REGION Network 96: CONTADOR DE PRESENCIA - CNT_pHsMx_E1E3
   RUNG wire#powerrail
      #CNT_pHsMx_E1E3(IN := wire#w4, R := wire#w7, PV := #V_CNT_pHsMx_E1, BaseUnidades_ms := "CTE_BaseUnidades_1ms", QU =>, QD =>, CVU =>, CVD =>)
   END_RUNG
   RUNG wire#powerrail
      Contact( #Mx_ET10 )
      wire#w1
      Contact( #CNTSeg_pHsMx_E1E3.QU )
      wire#w2
      Contact( #Selec_M1_Entrada )
      Contact( #pHsMx_2 )
      wire#w3
      Contact( #Avance_E1_Tx_Ok )
      I_Contact( #EstadoZona.Manual_CBx )
   END_RUNG wire#w4
   RUNG wire#powerrail
      Contact( #Mx_ET51 )
      Contact( #Simultaneo_Mx )
   END_RUNG wire#w1
   RUNG wire#powerrail
      Contact( #Mx_ET11 )
   END_RUNG wire#w2
   RUNG wire#powerrail
      Contact( #Mx_ET12 )
   END_RUNG wire#w2
   RUNG wire#w2
      Contact( #Selec_M3_Entrada )
      Contact( #pHsMx_1 )
   END_RUNG wire#w3
   RUNG wire#powerrail
      I_Contact( #Mx_ET10 )
      wire#w5
      I_Contact( #Mx_ET11 )
      I_Contact( #Mx_ET12 )
      wire#w6
      I_Contact( #Mx_ET51 )
   END_RUNG wire#w7
   RUNG wire#powerrail
      I_Contact( #CNTSeg_pHsMx_E1E3.QU )
   END_RUNG wire#w5
   RUNG wire#w6
      I_Contact( #CNTSeg_pHsMx_E1E3.QU )
   END_RUNG wire#w7
   RUNG wire#w6
      I_Contact( #Simultaneo_Mx )
   END_RUNG wire#w7
   // the same network as SCL:
   #CNT_pHsMx_E1E3(IN := (((#Mx_ET10 OR (#Mx_ET51 AND #Simultaneo_Mx)) AND #CNTSeg_pHsMx_E1E3.QU) OR #Mx_ET11 OR #Mx_ET12) AND ((#Selec_M1_Entrada AND #pHsMx_2) OR (#Selec_M3_Entrada AND #pHsMx_1)) AND #Avance_E1_Tx_Ok AND NOT #EstadoZona.Manual_CBx,   // "FB910_CNT_UHS"
                   R := (NOT #Mx_ET10 OR NOT #CNTSeg_pHsMx_E1E3.QU) AND NOT #Mx_ET11 AND NOT #Mx_ET12 AND (NOT #Mx_ET51 OR NOT #CNTSeg_pHsMx_E1E3.QU OR NOT #Simultaneo_Mx),
                   PV := #V_CNT_pHsMx_E1,
                   BaseUnidades_ms := "CTE_BaseUnidades_1ms");
END_REGION

REGION Network 97: DETERMINA PASO ET10 - ET11 (Nota: Control de Tiempo para dar el FTF a la Mesa Anterior)
   RUNG wire#powerrail
      I_Contact( #Mx_ET00 )
      { S7_Templates := "SrcType := Int" } LE_Contact(in1 := #CNT_pHsMx_E1E3.CVD, in2 := #V_CNT_pHsMx_FTF_E1)
      { S7_Templates := "SrcType := Int" } LT_Contact(in1 := #CNT_pHsMx_E1E3.CVD, in2 := #V_CNT_pHsMx_E1)
      wire#w1
      Contact( #Selec_M1_Entrada )
      Contact( #pHsMx_2 )
      wire#w2
      Coil( #CNT_pHsMx_FTF_OK_E1E3 )
   END_RUNG
   RUNG wire#w1
      Contact( #Selec_M3_Entrada )
      Contact( #pHsMx_1 )
   END_RUNG wire#w2
   // the same network as SCL:
   #CNT_pHsMx_FTF_OK_E1E3 := NOT #Mx_ET00 AND (#CNT_pHsMx_E1E3.CVD <= #V_CNT_pHsMx_FTF_E1) AND (#CNT_pHsMx_E1E3.CVD < #V_CNT_pHsMx_E1) AND ((#Selec_M1_Entrada AND #pHsMx_2) OR (#Selec_M3_Entrada AND #pHsMx_1));
END_REGION

REGION Network 98: CONTADOR DE SEGURIDAD DE PRESENCIA - CNTSeg_pHsMx_E2E4
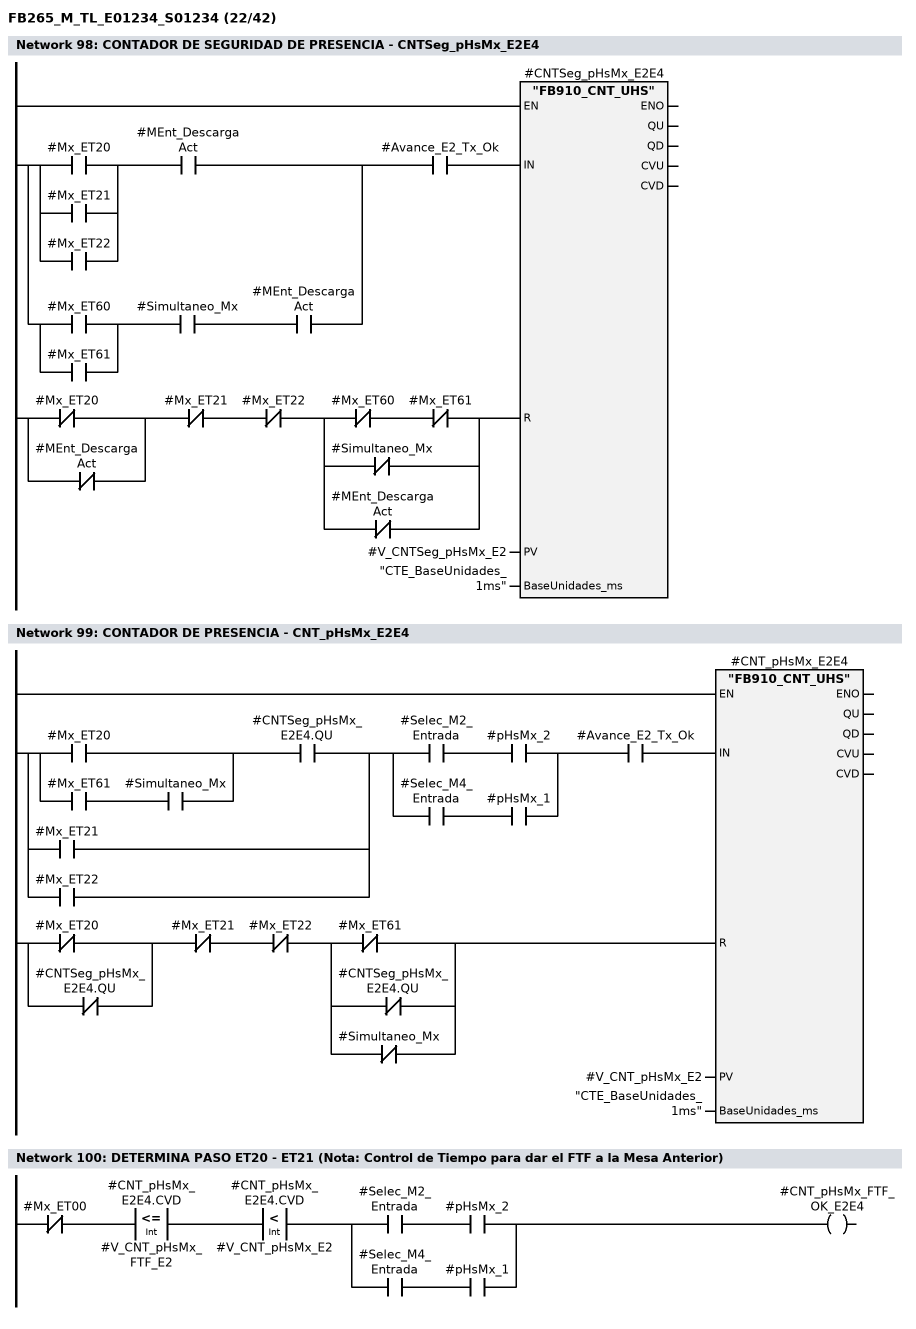
   RUNG wire#powerrail
      #CNTSeg_pHsMx_E2E4(IN := wire#w4, R := wire#w7, PV := #V_CNTSeg_pHsMx_E2, BaseUnidades_ms := "CTE_BaseUnidades_1ms", QU =>, QD =>, CVU =>, CVD =>)
   END_RUNG
   RUNG wire#powerrail
      Contact( #Mx_ET20 )
      wire#w1
      Contact( #MEnt_DescargaAct )
      wire#w2
      Contact( #Avance_E2_Tx_Ok )
   END_RUNG wire#w4
   RUNG wire#powerrail
      Contact( #Mx_ET21 )
   END_RUNG wire#w1
   RUNG wire#powerrail
      Contact( #Mx_ET22 )
   END_RUNG wire#w1
   RUNG wire#powerrail
      Contact( #Mx_ET60 )
      wire#w3
      Contact( #Simultaneo_Mx )
      Contact( #MEnt_DescargaAct )
   END_RUNG wire#w2
   RUNG wire#powerrail
      Contact( #Mx_ET61 )
   END_RUNG wire#w3
   RUNG wire#powerrail
      I_Contact( #Mx_ET20 )
      wire#w5
      I_Contact( #Mx_ET21 )
      I_Contact( #Mx_ET22 )
      wire#w6
      I_Contact( #Mx_ET60 )
      I_Contact( #Mx_ET61 )
   END_RUNG wire#w7
   RUNG wire#powerrail
      I_Contact( #MEnt_DescargaAct )
   END_RUNG wire#w5
   RUNG wire#w6
      I_Contact( #Simultaneo_Mx )
   END_RUNG wire#w7
   RUNG wire#w6
      I_Contact( #MEnt_DescargaAct )
   END_RUNG wire#w7
   // the same network as SCL:
   #CNTSeg_pHsMx_E2E4(IN := (((#Mx_ET20 OR #Mx_ET21 OR #Mx_ET22) AND #MEnt_DescargaAct) OR ((#Mx_ET60 OR #Mx_ET61) AND #Simultaneo_Mx AND #MEnt_DescargaAct)) AND #Avance_E2_Tx_Ok,   // "FB910_CNT_UHS"
                      R := (NOT #Mx_ET20 OR NOT #MEnt_DescargaAct) AND NOT #Mx_ET21 AND NOT #Mx_ET22 AND ((NOT #Mx_ET60 AND NOT #Mx_ET61) OR NOT #Simultaneo_Mx OR NOT #MEnt_DescargaAct),
                      PV := #V_CNTSeg_pHsMx_E2,
                      BaseUnidades_ms := "CTE_BaseUnidades_1ms");
END_REGION

REGION Network 99: CONTADOR DE PRESENCIA - CNT_pHsMx_E2E4
   RUNG wire#powerrail
      #CNT_pHsMx_E2E4(IN := wire#w4, R := wire#w7, PV := #V_CNT_pHsMx_E2, BaseUnidades_ms := "CTE_BaseUnidades_1ms", QU =>, QD =>, CVU =>, CVD =>)
   END_RUNG
   RUNG wire#powerrail
      Contact( #Mx_ET20 )
      wire#w1
      Contact( #CNTSeg_pHsMx_E2E4.QU )
      wire#w2
      Contact( #Selec_M2_Entrada )
      Contact( #pHsMx_2 )
      wire#w3
      Contact( #Avance_E2_Tx_Ok )
   END_RUNG wire#w4
   RUNG wire#powerrail
      Contact( #Mx_ET61 )
      Contact( #Simultaneo_Mx )
   END_RUNG wire#w1
   RUNG wire#powerrail
      Contact( #Mx_ET21 )
   END_RUNG wire#w2
   RUNG wire#powerrail
      Contact( #Mx_ET22 )
   END_RUNG wire#w2
   RUNG wire#w2
      Contact( #Selec_M4_Entrada )
      Contact( #pHsMx_1 )
   END_RUNG wire#w3
   RUNG wire#powerrail
      I_Contact( #Mx_ET20 )
      wire#w5
      I_Contact( #Mx_ET21 )
      I_Contact( #Mx_ET22 )
      wire#w6
      I_Contact( #Mx_ET61 )
   END_RUNG wire#w7
   RUNG wire#powerrail
      I_Contact( #CNTSeg_pHsMx_E2E4.QU )
   END_RUNG wire#w5
   RUNG wire#w6
      I_Contact( #CNTSeg_pHsMx_E2E4.QU )
   END_RUNG wire#w7
   RUNG wire#w6
      I_Contact( #Simultaneo_Mx )
   END_RUNG wire#w7
   // the same network as SCL:
   #CNT_pHsMx_E2E4(IN := (((#Mx_ET20 OR (#Mx_ET61 AND #Simultaneo_Mx)) AND #CNTSeg_pHsMx_E2E4.QU) OR #Mx_ET21 OR #Mx_ET22) AND ((#Selec_M2_Entrada AND #pHsMx_2) OR (#Selec_M4_Entrada AND #pHsMx_1)) AND #Avance_E2_Tx_Ok,   // "FB910_CNT_UHS"
                   R := (NOT #Mx_ET20 OR NOT #CNTSeg_pHsMx_E2E4.QU) AND NOT #Mx_ET21 AND NOT #Mx_ET22 AND (NOT #Mx_ET61 OR NOT #CNTSeg_pHsMx_E2E4.QU OR NOT #Simultaneo_Mx),
                   PV := #V_CNT_pHsMx_E2,
                   BaseUnidades_ms := "CTE_BaseUnidades_1ms");
END_REGION

REGION Network 100: DETERMINA PASO ET20 - ET21 (Nota: Control de Tiempo para dar el FTF a la Mesa Anterior)
   RUNG wire#powerrail
      I_Contact( #Mx_ET00 )
      { S7_Templates := "SrcType := Int" } LE_Contact(in1 := #CNT_pHsMx_E2E4.CVD, in2 := #V_CNT_pHsMx_FTF_E2)
      { S7_Templates := "SrcType := Int" } LT_Contact(in1 := #CNT_pHsMx_E2E4.CVD, in2 := #V_CNT_pHsMx_E2)
      wire#w1
      Contact( #Selec_M2_Entrada )
      Contact( #pHsMx_2 )
      wire#w2
      Coil( #CNT_pHsMx_FTF_OK_E2E4 )
   END_RUNG
   RUNG wire#w1
      Contact( #Selec_M4_Entrada )
      Contact( #pHsMx_1 )
   END_RUNG wire#w2
   // the same network as SCL:
   #CNT_pHsMx_FTF_OK_E2E4 := NOT #Mx_ET00 AND (#CNT_pHsMx_E2E4.CVD <= #V_CNT_pHsMx_FTF_E2) AND (#CNT_pHsMx_E2E4.CVD < #V_CNT_pHsMx_E2) AND ((#Selec_M2_Entrada AND #pHsMx_2) OR (#Selec_M4_Entrada AND #pHsMx_1));
END_REGION

REGION Network 101: CONTADOR SEGURIDAD DE AUSENCIA - CNTSeg_ApHsMx ??????? RESTAR VALOR DE POSICIONAMIENTO
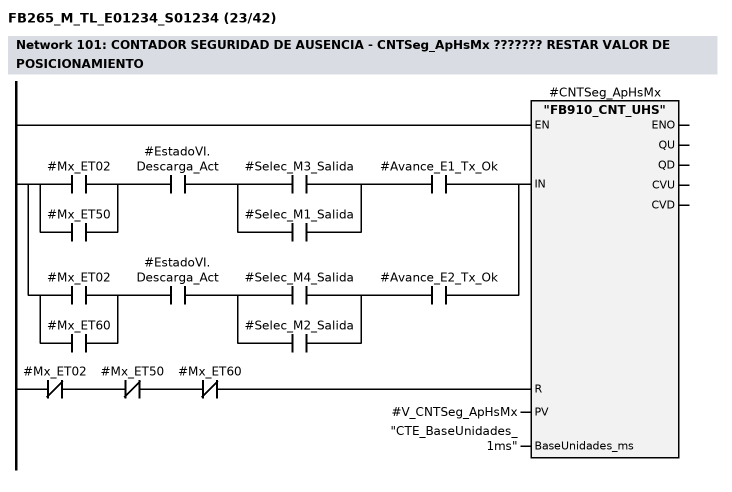
   RUNG wire#powerrail
      #CNTSeg_ApHsMx(IN := wire#w7, R := wire#w8, PV := #V_CNTSeg_ApHsMx, BaseUnidades_ms := "CTE_BaseUnidades_1ms", QU =>, QD =>, CVU =>, CVD =>)
   END_RUNG
   RUNG wire#powerrail
      Contact( #Mx_ET02 )
      wire#w1
      Contact( #EstadoVI.Descarga_Act )
      wire#w2
      Contact( #Selec_M3_Salida )
      wire#w3
      Contact( #Avance_E1_Tx_Ok )
   END_RUNG wire#w7
   RUNG wire#powerrail
      Contact( #Mx_ET50 )
   END_RUNG wire#w1
   RUNG wire#w2
      Contact( #Selec_M1_Salida )
   END_RUNG wire#w3
   RUNG wire#powerrail
      Contact( #Mx_ET02 )
      wire#w4
      Contact( #EstadoVI.Descarga_Act )
      wire#w5
      Contact( #Selec_M4_Salida )
      wire#w6
      Contact( #Avance_E2_Tx_Ok )
   END_RUNG wire#w7
   RUNG wire#powerrail
      Contact( #Mx_ET60 )
   END_RUNG wire#w4
   RUNG wire#w5
      Contact( #Selec_M2_Salida )
   END_RUNG wire#w6
   RUNG wire#powerrail
      I_Contact( #Mx_ET02 )
      I_Contact( #Mx_ET50 )
      I_Contact( #Mx_ET60 )
   END_RUNG wire#w8
   // the same network as SCL:
   #CNTSeg_ApHsMx(IN := ((#Mx_ET02 OR #Mx_ET50) AND #EstadoVI.Descarga_Act AND (#Selec_M3_Salida OR #Selec_M1_Salida) AND #Avance_E1_Tx_Ok) OR ((#Mx_ET02 OR #Mx_ET60) AND #EstadoVI.Descarga_Act AND (#Selec_M4_Salida OR #Selec_M2_Salida) AND #Avance_E2_Tx_Ok),   // "FB910_CNT_UHS"
                  R := NOT #Mx_ET02 AND NOT #Mx_ET50 AND NOT #Mx_ET60,
                  PV := #V_CNTSeg_ApHsMx,
                  BaseUnidades_ms := "CTE_BaseUnidades_1ms");
END_REGION

REGION Network 102: CONTADOR DE LA AUSENCIA - CNT_ApHsMX
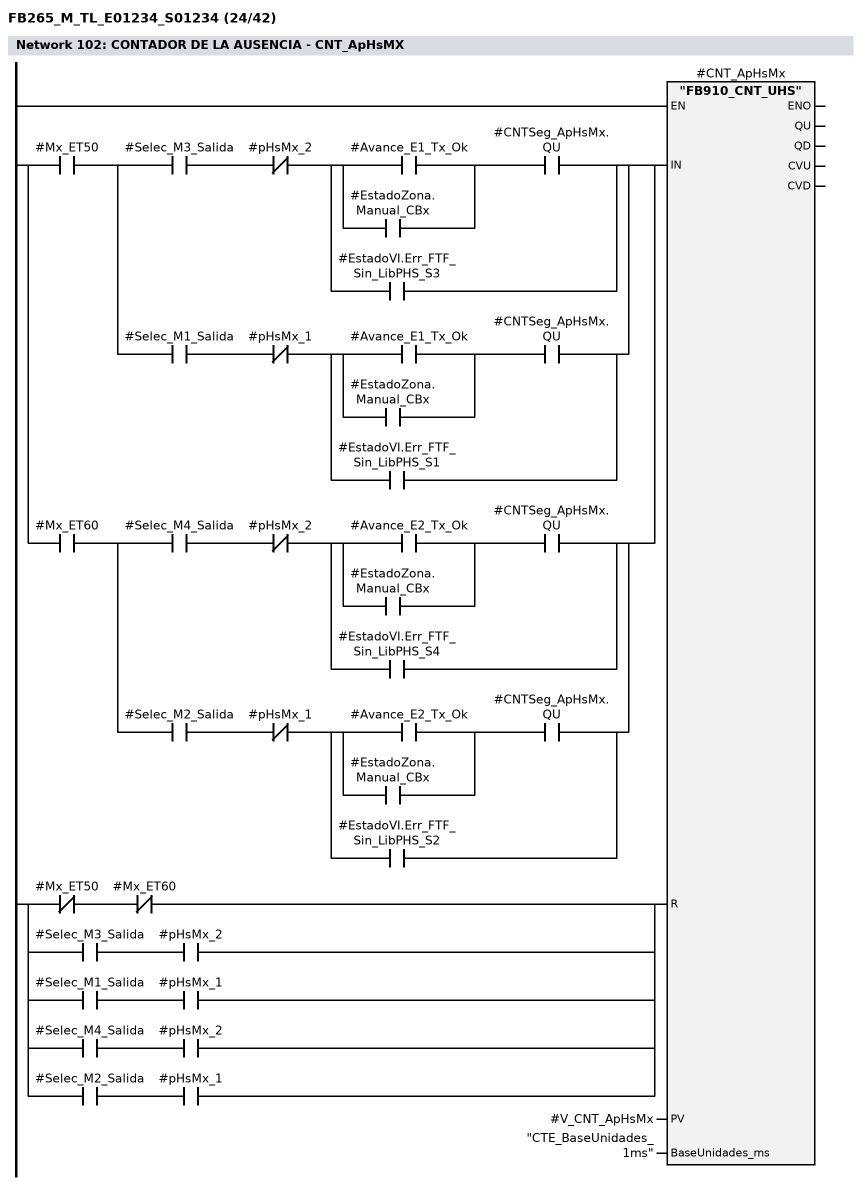
   RUNG wire#powerrail
      #CNT_ApHsMx(IN := wire#w11, R := wire#w12, PV := #V_CNT_ApHsMx, BaseUnidades_ms := "CTE_BaseUnidades_1ms", QU =>, QD =>, CVU =>, CVD =>)
   END_RUNG
   RUNG wire#powerrail
      Contact( #Mx_ET50 )
      wire#w1
      Contact( #Selec_M3_Salida )
      I_Contact( #pHsMx_2 )
      wire#w2
      Contact( #Avance_E1_Tx_Ok )
      wire#w3
      Contact( #CNTSeg_ApHsMx.QU )
   END_RUNG wire#w11
   RUNG wire#w2
      Contact( #EstadoZona.Manual_CBx )
   END_RUNG wire#w3
   RUNG wire#w2
      Contact( #EstadoVI.Err_FTF_Sin_LibPHS_S3 )
   END_RUNG wire#w11
   RUNG wire#w1
      Contact( #Selec_M1_Salida )
      I_Contact( #pHsMx_1 )
      wire#w4
      Contact( #Avance_E1_Tx_Ok )
      wire#w5
      Contact( #CNTSeg_ApHsMx.QU )
   END_RUNG wire#w11
   RUNG wire#w4
      Contact( #EstadoZona.Manual_CBx )
   END_RUNG wire#w5
   RUNG wire#w4
      Contact( #EstadoVI.Err_FTF_Sin_LibPHS_S1 )
   END_RUNG wire#w11
   RUNG wire#powerrail
      Contact( #Mx_ET60 )
      wire#w6
      Contact( #Selec_M4_Salida )
      I_Contact( #pHsMx_2 )
      wire#w7
      Contact( #Avance_E2_Tx_Ok )
      wire#w8
      Contact( #CNTSeg_ApHsMx.QU )
   END_RUNG wire#w11
   RUNG wire#w7
      Contact( #EstadoZona.Manual_CBx )
   END_RUNG wire#w8
   RUNG wire#w7
      Contact( #EstadoVI.Err_FTF_Sin_LibPHS_S4 )
   END_RUNG wire#w11
   RUNG wire#w6
      Contact( #Selec_M2_Salida )
      I_Contact( #pHsMx_1 )
      wire#w9
      Contact( #Avance_E2_Tx_Ok )
      wire#w10
      Contact( #CNTSeg_ApHsMx.QU )
   END_RUNG wire#w11
   RUNG wire#w9
      Contact( #EstadoZona.Manual_CBx )
   END_RUNG wire#w10
   RUNG wire#w9
      Contact( #EstadoVI.Err_FTF_Sin_LibPHS_S2 )
   END_RUNG wire#w11
   RUNG wire#powerrail
      I_Contact( #Mx_ET50 )
      I_Contact( #Mx_ET60 )
   END_RUNG wire#w12
   RUNG wire#powerrail
      Contact( #Selec_M3_Salida )
      Contact( #pHsMx_2 )
   END_RUNG wire#w12
   RUNG wire#powerrail
      Contact( #Selec_M1_Salida )
      Contact( #pHsMx_1 )
   END_RUNG wire#w12
   RUNG wire#powerrail
      Contact( #Selec_M4_Salida )
      Contact( #pHsMx_2 )
   END_RUNG wire#w12
   RUNG wire#powerrail
      Contact( #Selec_M2_Salida )
      Contact( #pHsMx_1 )
   END_RUNG wire#w12
   // the same network as SCL:
   #CNT_ApHsMx(IN := (#Mx_ET50 AND ((#Selec_M3_Salida AND NOT #pHsMx_2 AND (((#Avance_E1_Tx_Ok OR #EstadoZona.Manual_CBx) AND #CNTSeg_ApHsMx.QU) OR #EstadoVI.Err_FTF_Sin_LibPHS_S3)) OR (#Selec_M1_Salida AND NOT #pHsMx_1 AND (((#Avance_E1_Tx_Ok OR #EstadoZona.Manual_CBx) AND #CNTSeg_ApHsMx.QU) OR #EstadoVI.Err_FTF_Sin_LibPHS_S1)))) OR (#Mx_ET60 AND ((#Selec_M4_Salida AND NOT #pHsMx_2 AND (((#Avance_E2_Tx_Ok OR #EstadoZona.Manual_CBx) AND #CNTSeg_ApHsMx.QU) OR #EstadoVI.Err_FTF_Sin_LibPHS_S4)) OR (#Selec_M2_Salida AND NOT #pHsMx_1 AND (((#Avance_E2_Tx_Ok OR #EstadoZona.Manual_CBx) AND #CNTSeg_ApHsMx.QU) OR #EstadoVI.Err_FTF_Sin_LibPHS_S2)))),   // "FB910_CNT_UHS"
               R := (NOT #Mx_ET50 AND NOT #Mx_ET60) OR (#Selec_M3_Salida AND #pHsMx_2) OR (#Selec_M1_Salida AND #pHsMx_1) OR (#Selec_M4_Salida AND #pHsMx_2) OR (#Selec_M2_Salida AND #pHsMx_1),
               PV := #V_CNT_ApHsMx,
               BaseUnidades_ms := "CTE_BaseUnidades_1ms");
END_REGION

REGION Network 103: TEMPORIZADOR DE BLOQUEO DE MESA
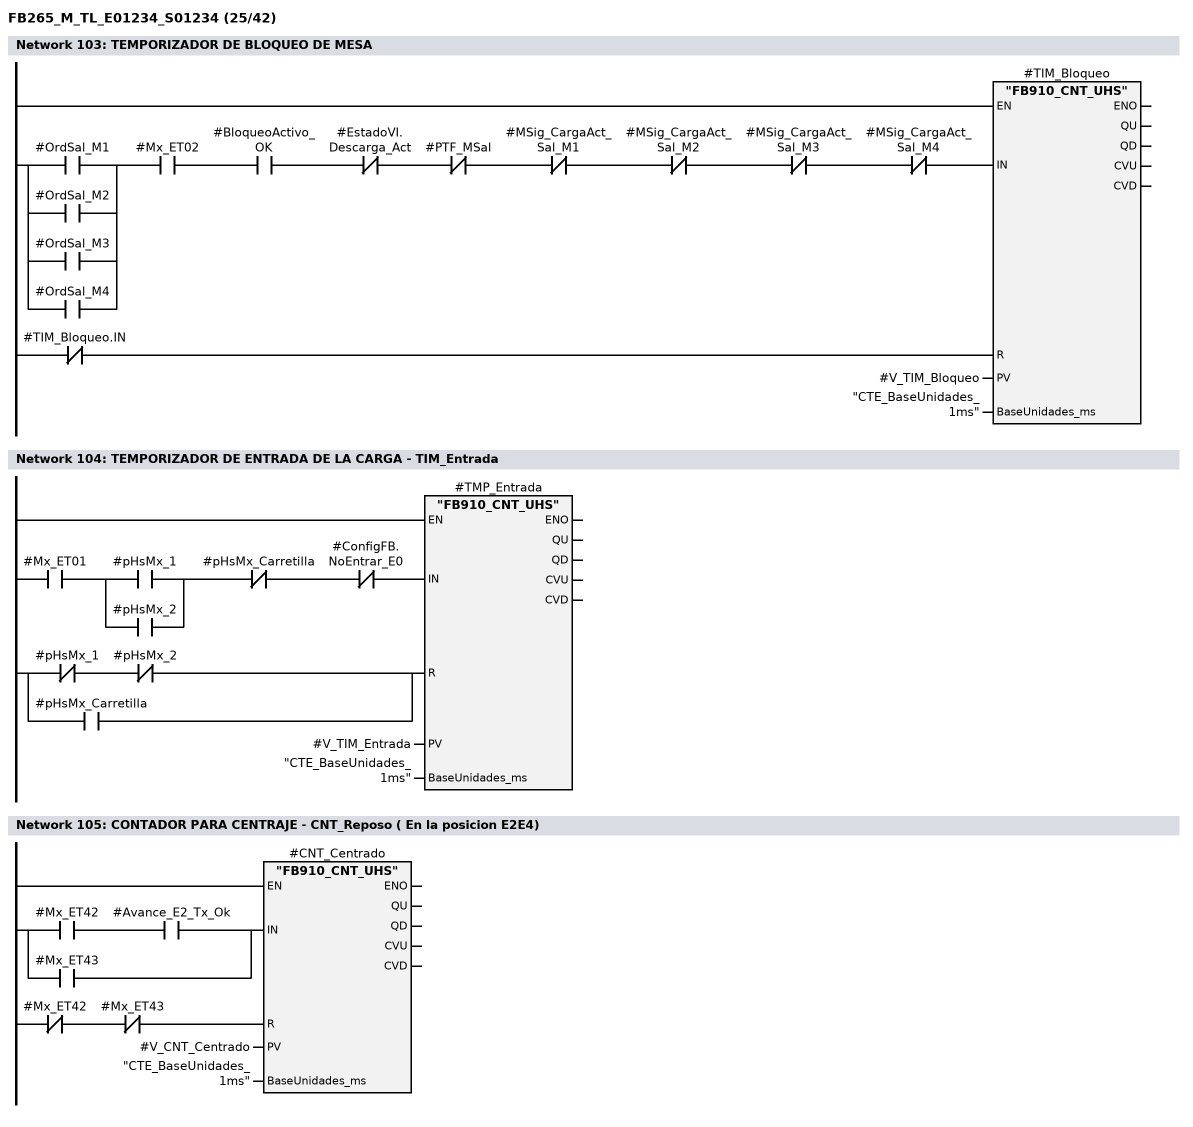
   RUNG wire#powerrail
      #TIM_Bloqueo(IN := wire#w2, R := wire#w3, PV := #V_TIM_Bloqueo, BaseUnidades_ms := "CTE_BaseUnidades_1ms", QU =>, QD =>, CVU =>, CVD =>)
   END_RUNG
   RUNG wire#powerrail
      Contact( #OrdSal_M1 )
      wire#w1
      Contact( #Mx_ET02 )
      Contact( #BloqueoActivo_OK )
      I_Contact( #EstadoVI.Descarga_Act )
      I_Contact( #PTF_MSal )
      I_Contact( #MSig_CargaAct_Sal_M1 )
      I_Contact( #MSig_CargaAct_Sal_M2 )
      I_Contact( #MSig_CargaAct_Sal_M3 )
      I_Contact( #MSig_CargaAct_Sal_M4 )
   END_RUNG wire#w2
   RUNG wire#powerrail
      Contact( #OrdSal_M2 )
   END_RUNG wire#w1
   RUNG wire#powerrail
      Contact( #OrdSal_M3 )
   END_RUNG wire#w1
   RUNG wire#powerrail
      Contact( #OrdSal_M4 )
   END_RUNG wire#w1
   RUNG wire#powerrail
      I_Contact( #TIM_Bloqueo.IN )
   END_RUNG wire#w3
   // the same network as SCL:
   #TIM_Bloqueo(IN := (#OrdSal_M1 OR #OrdSal_M2 OR #OrdSal_M3 OR #OrdSal_M4) AND #Mx_ET02 AND #BloqueoActivo_OK AND NOT #EstadoVI.Descarga_Act AND NOT #PTF_MSal AND NOT #MSig_CargaAct_Sal_M1 AND NOT #MSig_CargaAct_Sal_M2 AND NOT #MSig_CargaAct_Sal_M3 AND NOT #MSig_CargaAct_Sal_M4,   // "FB910_CNT_UHS"
                R := NOT #TIM_Bloqueo.IN,
                PV := #V_TIM_Bloqueo,
                BaseUnidades_ms := "CTE_BaseUnidades_1ms");
END_REGION

REGION Network 104: TEMPORIZADOR DE ENTRADA DE LA CARGA - TIM_Entrada
   RUNG wire#powerrail
      #TMP_Entrada(IN := wire#w3, R := wire#w4, PV := #V_TIM_Entrada, BaseUnidades_ms := "CTE_BaseUnidades_1ms", QU =>, QD =>, CVU =>, CVD =>)
   END_RUNG
   RUNG wire#powerrail
      Contact( #Mx_ET01 )
      wire#w1
      Contact( #pHsMx_1 )
      wire#w2
      I_Contact( #pHsMx_Carretilla )
      I_Contact( #ConfigFB.NoEntrar_E0 )
   END_RUNG wire#w3
   RUNG wire#w1
      Contact( #pHsMx_2 )
   END_RUNG wire#w2
   RUNG wire#powerrail
      I_Contact( #pHsMx_1 )
      I_Contact( #pHsMx_2 )
   END_RUNG wire#w4
   RUNG wire#powerrail
      Contact( #pHsMx_Carretilla )
   END_RUNG wire#w4
   // the same network as SCL:
   #TMP_Entrada(IN := #Mx_ET01 AND (#pHsMx_1 OR #pHsMx_2) AND NOT #pHsMx_Carretilla AND NOT #ConfigFB.NoEntrar_E0,   // "FB910_CNT_UHS"
                R := (NOT #pHsMx_1 AND NOT #pHsMx_2) OR #pHsMx_Carretilla,
                PV := #V_TIM_Entrada,
                BaseUnidades_ms := "CTE_BaseUnidades_1ms");
END_REGION

REGION Network 105: CONTADOR PARA CENTRAJE - CNT_Reposo ( En la posicion E2E4)
   RUNG wire#powerrail
      #CNT_Centrado(IN := wire#w1, R := wire#w2, PV := #V_CNT_Centrado, BaseUnidades_ms := "CTE_BaseUnidades_1ms", QU =>, QD =>, CVU =>, CVD =>)
   END_RUNG
   RUNG wire#powerrail
      Contact( #Mx_ET42 )
      Contact( #Avance_E2_Tx_Ok )
   END_RUNG wire#w1
   RUNG wire#powerrail
      Contact( #Mx_ET43 )
   END_RUNG wire#w1
   RUNG wire#powerrail
      I_Contact( #Mx_ET42 )
      I_Contact( #Mx_ET43 )
   END_RUNG wire#w2
   // the same network as SCL:
   #CNT_Centrado(IN := (#Mx_ET42 AND #Avance_E2_Tx_Ok) OR #Mx_ET43,   // "FB910_CNT_UHS"
                 R := NOT #Mx_ET42 AND NOT #Mx_ET43,
                 PV := #V_CNT_Centrado,
                 BaseUnidades_ms := "CTE_BaseUnidades_1ms");
END_REGION

REGION Network 106: TEMPORIZADOR DE RETIRADA DE LA CARGA - TIM_Salida
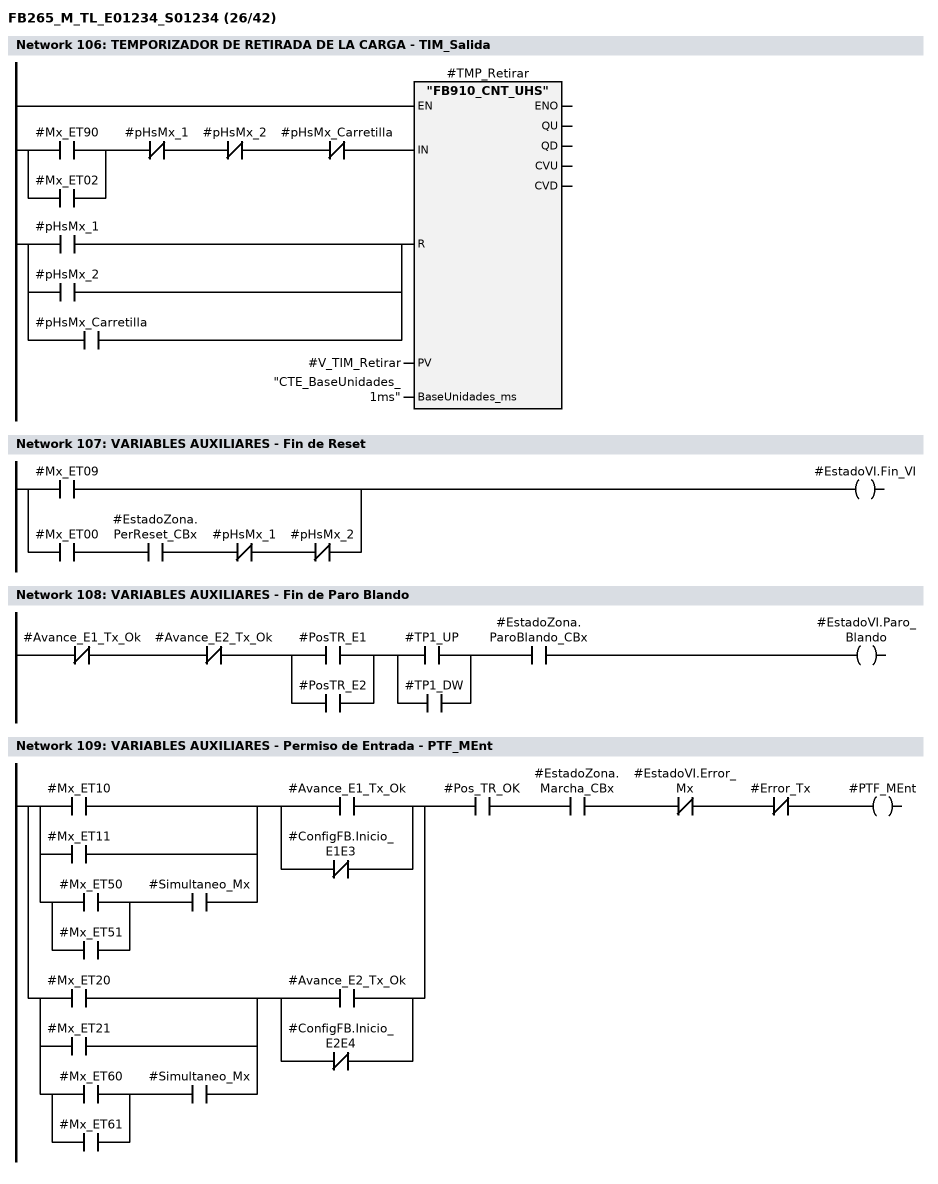
   RUNG wire#powerrail
      #TMP_Retirar(IN := wire#w2, R := wire#w3, PV := #V_TIM_Retirar, BaseUnidades_ms := "CTE_BaseUnidades_1ms", QU =>, QD =>, CVU =>, CVD =>)
   END_RUNG
   RUNG wire#powerrail
      Contact( #Mx_ET90 )
      wire#w1
      I_Contact( #pHsMx_1 )
      I_Contact( #pHsMx_2 )
      I_Contact( #pHsMx_Carretilla )
   END_RUNG wire#w2
   RUNG wire#powerrail
      Contact( #Mx_ET02 )
   END_RUNG wire#w1
   RUNG wire#powerrail
      Contact( #pHsMx_1 )
   END_RUNG wire#w3
   RUNG wire#powerrail
      Contact( #pHsMx_2 )
   END_RUNG wire#w3
   RUNG wire#powerrail
      Contact( #pHsMx_Carretilla )
   END_RUNG wire#w3
   // the same network as SCL:
   #TMP_Retirar(IN := (#Mx_ET90 OR #Mx_ET02) AND NOT #pHsMx_1 AND NOT #pHsMx_2 AND NOT #pHsMx_Carretilla,   // "FB910_CNT_UHS"
                R := #pHsMx_1 OR #pHsMx_2 OR #pHsMx_Carretilla,
                PV := #V_TIM_Retirar,
                BaseUnidades_ms := "CTE_BaseUnidades_1ms");
END_REGION

REGION Network 107: VARIABLES AUXILIARES - Fin de Reset
   RUNG wire#powerrail
      Contact( #Mx_ET09 )
      wire#w1
      Coil( #EstadoVI.Fin_VI )
   END_RUNG
   RUNG wire#powerrail
      Contact( #Mx_ET00 )
      Contact( #EstadoZona.PerReset_CBx )
      I_Contact( #pHsMx_1 )
      I_Contact( #pHsMx_2 )
   END_RUNG wire#w1
   // the same network as SCL:
   #EstadoVI.Fin_VI := #Mx_ET09 OR (#Mx_ET00 AND #EstadoZona.PerReset_CBx AND NOT #pHsMx_1 AND NOT #pHsMx_2);
END_REGION

REGION Network 108: VARIABLES AUXILIARES - Fin de Paro Blando
   RUNG wire#powerrail
      I_Contact( #Avance_E1_Tx_Ok )
      I_Contact( #Avance_E2_Tx_Ok )
      wire#w1
      Contact( #PosTR_E1 )
      wire#w2
      Contact( #TP1_UP )
      wire#w3
      Contact( #EstadoZona.ParoBlando_CBx )
      Coil( #EstadoVI.Paro_Blando )
   END_RUNG
   RUNG wire#w1
      Contact( #PosTR_E2 )
   END_RUNG wire#w2
   RUNG wire#w2
      Contact( #TP1_DW )
   END_RUNG wire#w3
   // the same network as SCL:
   #EstadoVI.Paro_Blando := NOT #Avance_E1_Tx_Ok AND NOT #Avance_E2_Tx_Ok AND (#PosTR_E1 OR #PosTR_E2) AND (#TP1_UP OR #TP1_DW) AND #EstadoZona.ParoBlando_CBx;
END_REGION

REGION Network 109: VARIABLES AUXILIARES - Permiso de Entrada - PTF_MEnt
   RUNG wire#powerrail
      Contact( #Mx_ET10 )
      wire#w1
      Contact( #Avance_E1_Tx_Ok )
      wire#w3
      Contact( #Pos_TR_OK )
      Contact( #EstadoZona.Marcha_CBx )
      I_Contact( #EstadoVI.Error_Mx )
      I_Contact( #Error_Tx )
      Coil( #PTF_MEnt )
   END_RUNG
   RUNG wire#powerrail
      Contact( #Mx_ET11 )
   END_RUNG wire#w1
   RUNG wire#powerrail
      Contact( #Mx_ET50 )
      wire#w2
      Contact( #Simultaneo_Mx )
   END_RUNG wire#w1
   RUNG wire#powerrail
      Contact( #Mx_ET51 )
   END_RUNG wire#w2
   RUNG wire#w1
      I_Contact( #ConfigFB.Inicio_E1E3 )
   END_RUNG wire#w3
   RUNG wire#powerrail
      Contact( #Mx_ET20 )
      wire#w4
      Contact( #Avance_E2_Tx_Ok )
   END_RUNG wire#w3
   RUNG wire#powerrail
      Contact( #Mx_ET21 )
   END_RUNG wire#w4
   RUNG wire#powerrail
      Contact( #Mx_ET60 )
      wire#w5
      Contact( #Simultaneo_Mx )
   END_RUNG wire#w4
   RUNG wire#powerrail
      Contact( #Mx_ET61 )
   END_RUNG wire#w5
   RUNG wire#w4
      I_Contact( #ConfigFB.Inicio_E2E4 )
   END_RUNG wire#w3
   // the same network as SCL:
   #PTF_MEnt := (((#Mx_ET10 OR #Mx_ET11 OR ((#Mx_ET50 OR #Mx_ET51) AND #Simultaneo_Mx)) AND (#Avance_E1_Tx_Ok OR NOT #ConfigFB.Inicio_E1E3)) OR ((#Mx_ET20 OR #Mx_ET21 OR ((#Mx_ET60 OR #Mx_ET61) AND #Simultaneo_Mx)) AND (#Avance_E2_Tx_Ok OR NOT #ConfigFB.Inicio_E2E4))) AND #Pos_TR_OK AND #EstadoZona.Marcha_CBx AND NOT #EstadoVI.Error_Mx AND NOT #Error_Tx;
END_REGION

REGION Network 110: VARIABLES AUXILIARES - Aviso de Salida - AVTF_MSal
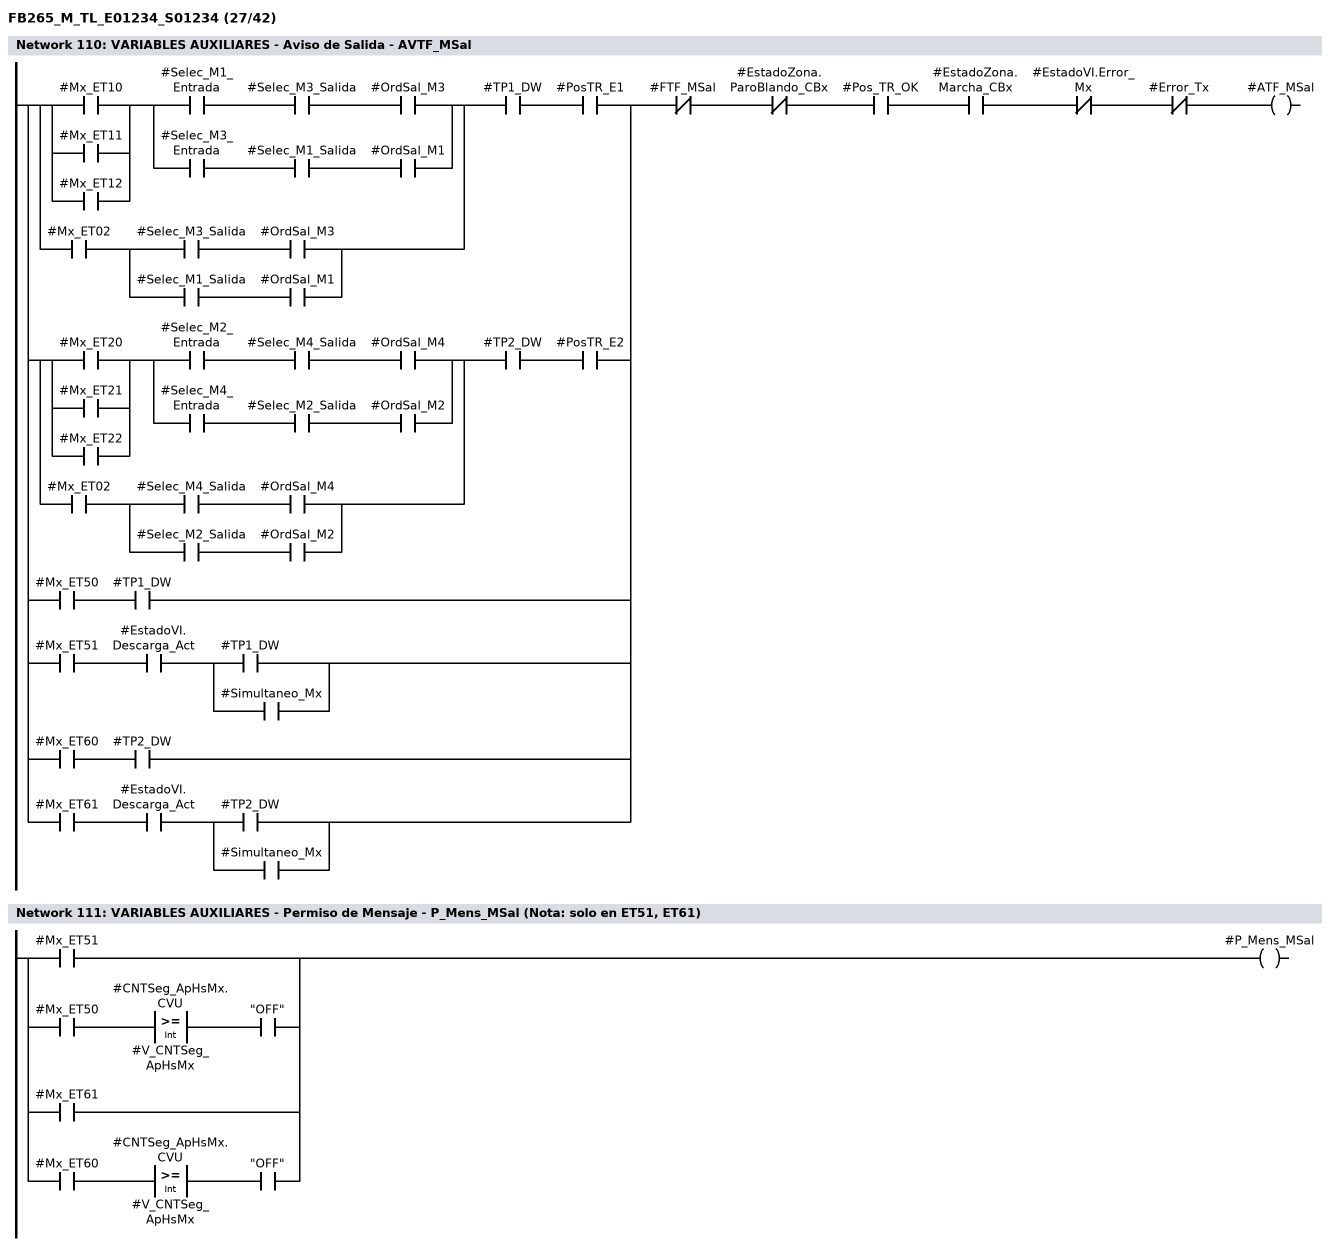
   RUNG wire#powerrail
      Contact( #Mx_ET10 )
      wire#w1
      Contact( #Selec_M1_Entrada )
      Contact( #Selec_M3_Salida )
      Contact( #OrdSal_M3 )
      wire#w2
      Contact( #TP1_DW )
      Contact( #PosTR_E1 )
      wire#w4
      I_Contact( #FTF_MSal )
      I_Contact( #EstadoZona.ParoBlando_CBx )
      Contact( #Pos_TR_OK )
      Contact( #EstadoZona.Marcha_CBx )
      I_Contact( #EstadoVI.Error_Mx )
      I_Contact( #Error_Tx )
      Coil( #ATF_MSal )
   END_RUNG
   RUNG wire#powerrail
      Contact( #Mx_ET11 )
   END_RUNG wire#w1
   RUNG wire#powerrail
      Contact( #Mx_ET12 )
   END_RUNG wire#w1
   RUNG wire#w1
      Contact( #Selec_M3_Entrada )
      Contact( #Selec_M1_Salida )
      Contact( #OrdSal_M1 )
   END_RUNG wire#w2
   RUNG wire#powerrail
      Contact( #Mx_ET02 )
      wire#w3
      Contact( #Selec_M3_Salida )
      Contact( #OrdSal_M3 )
   END_RUNG wire#w2
   RUNG wire#w3
      Contact( #Selec_M1_Salida )
      Contact( #OrdSal_M1 )
   END_RUNG wire#w2
   RUNG wire#powerrail
      Contact( #Mx_ET20 )
      wire#w5
      Contact( #Selec_M2_Entrada )
      Contact( #Selec_M4_Salida )
      Contact( #OrdSal_M4 )
      wire#w6
      Contact( #TP2_DW )
      Contact( #PosTR_E2 )
   END_RUNG wire#w4
   RUNG wire#powerrail
      Contact( #Mx_ET21 )
   END_RUNG wire#w5
   RUNG wire#powerrail
      Contact( #Mx_ET22 )
   END_RUNG wire#w5
   RUNG wire#w5
      Contact( #Selec_M4_Entrada )
      Contact( #Selec_M2_Salida )
      Contact( #OrdSal_M2 )
   END_RUNG wire#w6
   RUNG wire#powerrail
      Contact( #Mx_ET02 )
      wire#w7
      Contact( #Selec_M4_Salida )
      Contact( #OrdSal_M4 )
   END_RUNG wire#w6
   RUNG wire#w7
      Contact( #Selec_M2_Salida )
      Contact( #OrdSal_M2 )
   END_RUNG wire#w6
   RUNG wire#powerrail
      Contact( #Mx_ET50 )
      Contact( #TP1_DW )
   END_RUNG wire#w4
   RUNG wire#powerrail
      Contact( #Mx_ET51 )
      Contact( #EstadoVI.Descarga_Act )
      wire#w8
      Contact( #TP1_DW )
   END_RUNG wire#w4
   RUNG wire#w8
      Contact( #Simultaneo_Mx )
   END_RUNG wire#w4
   RUNG wire#powerrail
      Contact( #Mx_ET60 )
      Contact( #TP2_DW )
   END_RUNG wire#w4
   RUNG wire#powerrail
      Contact( #Mx_ET61 )
      Contact( #EstadoVI.Descarga_Act )
      wire#w9
      Contact( #TP2_DW )
   END_RUNG wire#w4
   RUNG wire#w9
      Contact( #Simultaneo_Mx )
   END_RUNG wire#w4
   // the same network as SCL:
   #ATF_MSal := (((((#Mx_ET10 OR #Mx_ET11 OR #Mx_ET12) AND ((#Selec_M1_Entrada AND #Selec_M3_Salida AND #OrdSal_M3) OR (#Selec_M3_Entrada AND #Selec_M1_Salida AND #OrdSal_M1))) OR (#Mx_ET02 AND ((#Selec_M3_Salida AND #OrdSal_M3) OR (#Selec_M1_Salida AND #OrdSal_M1)))) AND #TP1_DW AND #PosTR_E1) OR ((((#Mx_ET20 OR #Mx_ET21 OR #Mx_ET22) AND ((#Selec_M2_Entrada AND #Selec_M4_Salida AND #OrdSal_M4) OR (#Selec_M4_Entrada AND #Selec_M2_Salida AND #OrdSal_M2))) OR (#Mx_ET02 AND ((#Selec_M4_Salida AND #OrdSal_M4) OR (#Selec_M2_Salida AND #OrdSal_M2)))) AND #TP2_DW AND #PosTR_E2) OR (#Mx_ET50 AND #TP1_DW) OR (#Mx_ET51 AND #EstadoVI.Descarga_Act AND (#TP1_DW OR #Simultaneo_Mx)) OR (#Mx_ET60 AND #TP2_DW) OR (#Mx_ET61 AND #EstadoVI.Descarga_Act AND (#TP2_DW OR #Simultaneo_Mx))) AND NOT #FTF_MSal AND NOT #EstadoZona.ParoBlando_CBx AND #Pos_TR_OK AND #EstadoZona.Marcha_CBx AND NOT #EstadoVI.Error_Mx AND NOT #Error_Tx;
END_REGION

REGION Network 111: VARIABLES AUXILIARES - Permiso de Mensaje - P_Mens_MSal (Nota: solo en ET51, ET61)
   RUNG wire#powerrail
      Contact( #Mx_ET51 )
      wire#w1
      Coil( #P_Mens_MSal )
   END_RUNG
   RUNG wire#powerrail
      Contact( #Mx_ET50 )
      { S7_Templates := "SrcType := Int" } GE_Contact(in1 := #CNTSeg_ApHsMx.CVU, in2 := #V_CNTSeg_ApHsMx)
      Contact( "OFF" )
   END_RUNG wire#w1
   RUNG wire#powerrail
      Contact( #Mx_ET61 )
   END_RUNG wire#w1
   RUNG wire#powerrail
      Contact( #Mx_ET60 )
      { S7_Templates := "SrcType := Int" } GE_Contact(in1 := #CNTSeg_ApHsMx.CVU, in2 := #V_CNTSeg_ApHsMx)
      Contact( "OFF" )
   END_RUNG wire#w1
   // the same network as SCL:
   #P_Mens_MSal := #Mx_ET51 OR (#Mx_ET50 AND (#CNTSeg_ApHsMx.CVU >= #V_CNTSeg_ApHsMx) AND "OFF") OR #Mx_ET61 OR (#Mx_ET60 AND (#CNTSeg_ApHsMx.CVU >= #V_CNTSeg_ApHsMx) AND "OFF");
END_REGION

REGION Network 112: VARIABLES AUXILIARES - Demultiplexado Señales de Entrada a la Mesa --> PTF
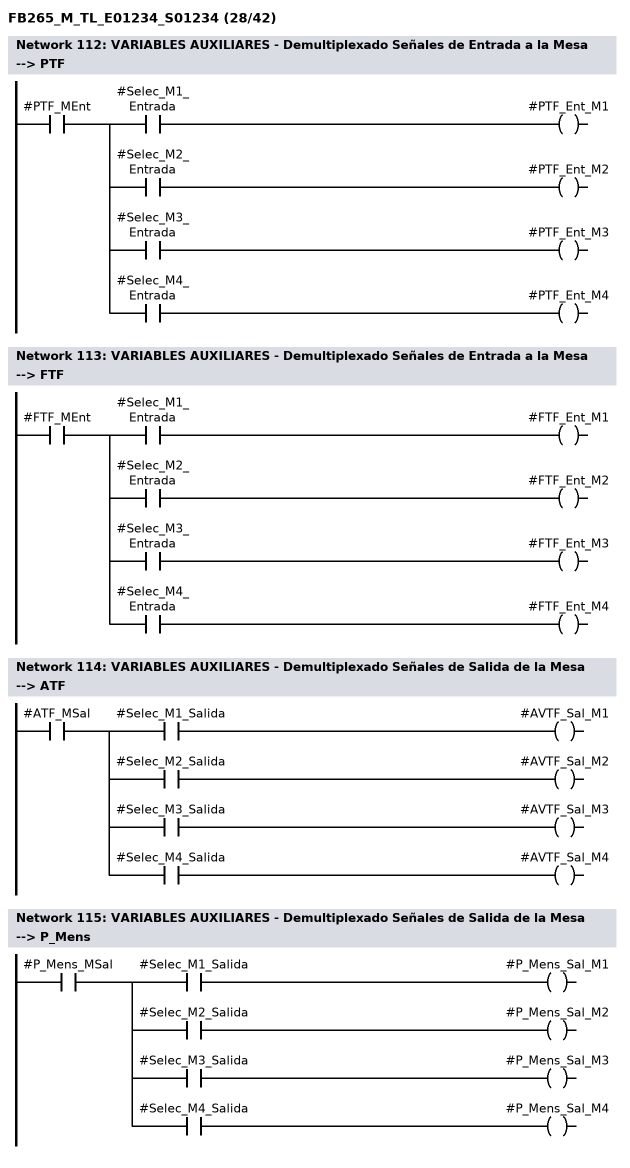
   RUNG wire#powerrail
      Contact( #PTF_MEnt )
      wire#w1
      Contact( #Selec_M1_Entrada )
      Coil( #PTF_Ent_M1 )
   END_RUNG
   RUNG wire#w1
      Contact( #Selec_M2_Entrada )
      Coil( #PTF_Ent_M2 )
   END_RUNG
   RUNG wire#w1
      Contact( #Selec_M3_Entrada )
      Coil( #PTF_Ent_M3 )
   END_RUNG
   RUNG wire#w1
      Contact( #Selec_M4_Entrada )
      Coil( #PTF_Ent_M4 )
   END_RUNG
   // the same network as SCL:
   #PTF_Ent_M1 := #PTF_MEnt AND #Selec_M1_Entrada;
   #PTF_Ent_M2 := #PTF_MEnt AND #Selec_M2_Entrada;
   #PTF_Ent_M3 := #PTF_MEnt AND #Selec_M3_Entrada;
   #PTF_Ent_M4 := #PTF_MEnt AND #Selec_M4_Entrada;
END_REGION

REGION Network 113: VARIABLES AUXILIARES - Demultiplexado Señales de Entrada a la Mesa --> FTF
   RUNG wire#powerrail
      Contact( #FTF_MEnt )
      wire#w1
      Contact( #Selec_M1_Entrada )
      Coil( #FTF_Ent_M1 )
   END_RUNG
   RUNG wire#w1
      Contact( #Selec_M2_Entrada )
      Coil( #FTF_Ent_M2 )
   END_RUNG
   RUNG wire#w1
      Contact( #Selec_M3_Entrada )
      Coil( #FTF_Ent_M3 )
   END_RUNG
   RUNG wire#w1
      Contact( #Selec_M4_Entrada )
      Coil( #FTF_Ent_M4 )
   END_RUNG
   // the same network as SCL:
   #FTF_Ent_M1 := #FTF_MEnt AND #Selec_M1_Entrada;
   #FTF_Ent_M2 := #FTF_MEnt AND #Selec_M2_Entrada;
   #FTF_Ent_M3 := #FTF_MEnt AND #Selec_M3_Entrada;
   #FTF_Ent_M4 := #FTF_MEnt AND #Selec_M4_Entrada;
END_REGION

REGION Network 114: VARIABLES AUXILIARES - Demultiplexado Señales de Salida de la Mesa --> ATF
   RUNG wire#powerrail
      Contact( #ATF_MSal )
      wire#w1
      Contact( #Selec_M1_Salida )
      Coil( #AVTF_Sal_M1 )
   END_RUNG
   RUNG wire#w1
      Contact( #Selec_M2_Salida )
      Coil( #AVTF_Sal_M2 )
   END_RUNG
   RUNG wire#w1
      Contact( #Selec_M3_Salida )
      Coil( #AVTF_Sal_M3 )
   END_RUNG
   RUNG wire#w1
      Contact( #Selec_M4_Salida )
      Coil( #AVTF_Sal_M4 )
   END_RUNG
   // the same network as SCL:
   #AVTF_Sal_M1 := #ATF_MSal AND #Selec_M1_Salida;
   #AVTF_Sal_M2 := #ATF_MSal AND #Selec_M2_Salida;
   #AVTF_Sal_M3 := #ATF_MSal AND #Selec_M3_Salida;
   #AVTF_Sal_M4 := #ATF_MSal AND #Selec_M4_Salida;
END_REGION

REGION Network 115: VARIABLES AUXILIARES - Demultiplexado Señales de Salida de la Mesa --> P_Mens
   RUNG wire#powerrail
      Contact( #P_Mens_MSal )
      wire#w1
      Contact( #Selec_M1_Salida )
      Coil( #P_Mens_Sal_M1 )
   END_RUNG
   RUNG wire#w1
      Contact( #Selec_M2_Salida )
      Coil( #P_Mens_Sal_M2 )
   END_RUNG
   RUNG wire#w1
      Contact( #Selec_M3_Salida )
      Coil( #P_Mens_Sal_M3 )
   END_RUNG
   RUNG wire#w1
      Contact( #Selec_M4_Salida )
      Coil( #P_Mens_Sal_M4 )
   END_RUNG
   // the same network as SCL:
   #P_Mens_Sal_M1 := #P_Mens_MSal AND #Selec_M1_Salida;
   #P_Mens_Sal_M2 := #P_Mens_MSal AND #Selec_M2_Salida;
   #P_Mens_Sal_M3 := #P_Mens_MSal AND #Selec_M3_Salida;
   #P_Mens_Sal_M4 := #P_Mens_MSal AND #Selec_M4_Salida;
END_REGION

REGION Network 116: CONTADOR DE SIMULTANEO
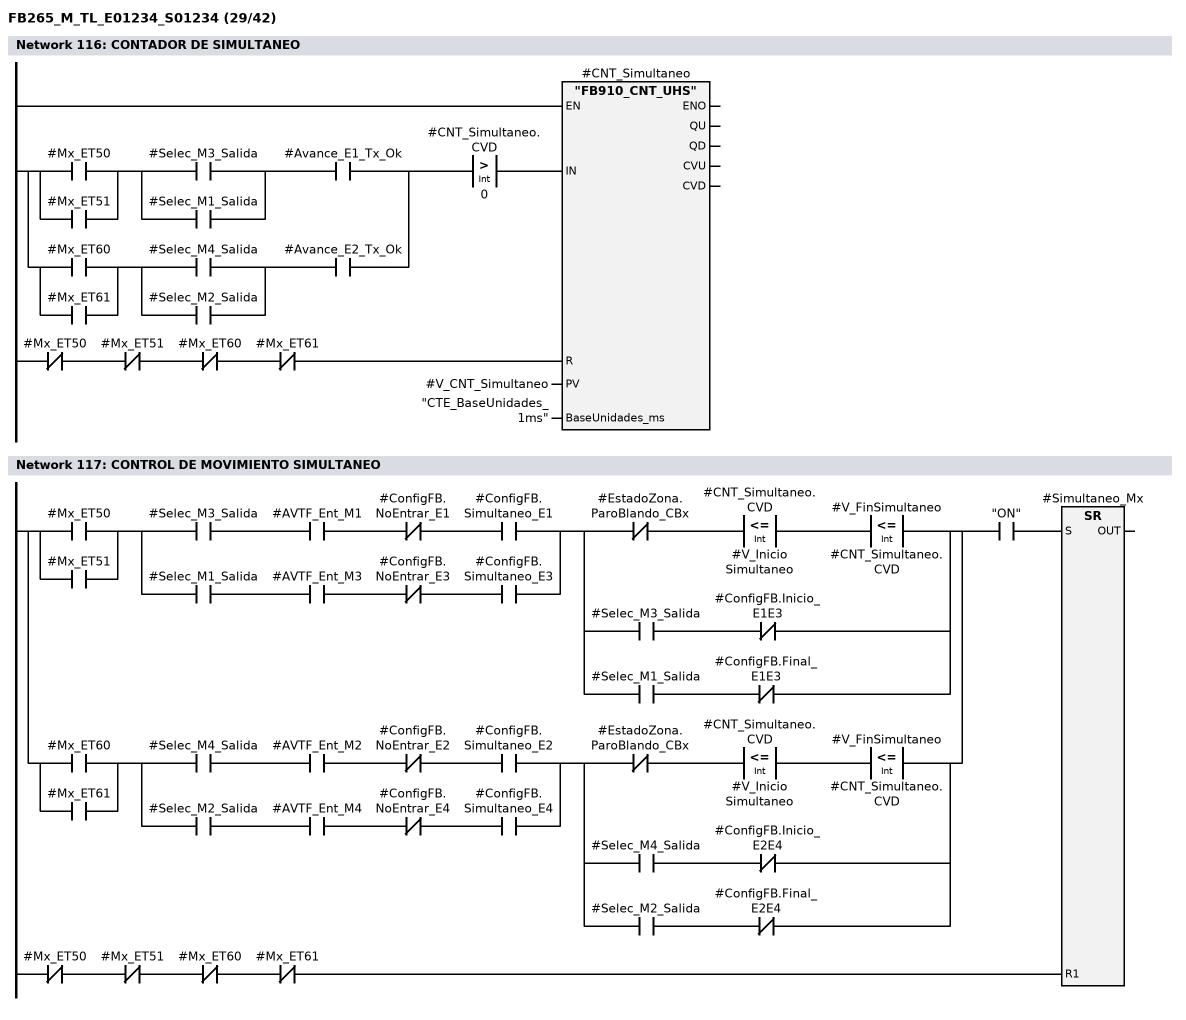
   RUNG wire#powerrail
      #CNT_Simultaneo(IN := wire#w6, R := wire#w7, PV := #V_CNT_Simultaneo, BaseUnidades_ms := "CTE_BaseUnidades_1ms", QU =>, QD =>, CVU =>, CVD =>)
   END_RUNG
   RUNG wire#powerrail
      Contact( #Mx_ET50 )
      wire#w1
      Contact( #Selec_M3_Salida )
      wire#w2
      Contact( #Avance_E1_Tx_Ok )
      wire#w3
      { S7_Templates := "SrcType := Int" } GT_Contact(in1 := #CNT_Simultaneo.CVD, in2 := 0)
   END_RUNG wire#w6
   RUNG wire#powerrail
      Contact( #Mx_ET51 )
   END_RUNG wire#w1
   RUNG wire#w1
      Contact( #Selec_M1_Salida )
   END_RUNG wire#w2
   RUNG wire#powerrail
      Contact( #Mx_ET60 )
      wire#w4
      Contact( #Selec_M4_Salida )
      wire#w5
      Contact( #Avance_E2_Tx_Ok )
   END_RUNG wire#w3
   RUNG wire#powerrail
      Contact( #Mx_ET61 )
   END_RUNG wire#w4
   RUNG wire#w4
      Contact( #Selec_M2_Salida )
   END_RUNG wire#w5
   RUNG wire#powerrail
      I_Contact( #Mx_ET50 )
      I_Contact( #Mx_ET51 )
      I_Contact( #Mx_ET60 )
      I_Contact( #Mx_ET61 )
   END_RUNG wire#w7
   // the same network as SCL:
   #CNT_Simultaneo(IN := (((#Mx_ET50 OR #Mx_ET51) AND (#Selec_M3_Salida OR #Selec_M1_Salida) AND #Avance_E1_Tx_Ok) OR ((#Mx_ET60 OR #Mx_ET61) AND (#Selec_M4_Salida OR #Selec_M2_Salida) AND #Avance_E2_Tx_Ok)) AND (#CNT_Simultaneo.CVD > 0),   // "FB910_CNT_UHS"
                   R := NOT #Mx_ET50 AND NOT #Mx_ET51 AND NOT #Mx_ET60 AND NOT #Mx_ET61,
                   PV := #V_CNT_Simultaneo,
                   BaseUnidades_ms := "CTE_BaseUnidades_1ms");
END_REGION

REGION Network 117: CONTROL DE MOVIMIENTO SIMULTANEO
   RUNG wire#powerrail
      Contact( #Mx_ET50 )
      wire#w1
      Contact( #Selec_M3_Salida )
      Contact( #AVTF_Ent_M1 )
      I_Contact( #ConfigFB.NoEntrar_E1 )
      Contact( #ConfigFB.Simultaneo_E1 )
      wire#w2
      I_Contact( #EstadoZona.ParoBlando_CBx )
      { S7_Templates := "SrcType := Int" } LE_Contact(in1 := #CNT_Simultaneo.CVD, in2 := #V_InicioSimultaneo)
      { S7_Templates := "SrcType := Int" } LE_Contact(in1 := #V_FinSimultaneo, in2 := #CNT_Simultaneo.CVD)
      wire#w3
      Contact( "ON" )
      S_SR(operand := #Simultaneo_Mx, r1 := wire#w6)
   END_RUNG
   RUNG wire#powerrail
      Contact( #Mx_ET51 )
   END_RUNG wire#w1
   RUNG wire#w1
      Contact( #Selec_M1_Salida )
      Contact( #AVTF_Ent_M3 )
      I_Contact( #ConfigFB.NoEntrar_E3 )
      Contact( #ConfigFB.Simultaneo_E3 )
   END_RUNG wire#w2
   RUNG wire#w2
      Contact( #Selec_M3_Salida )
      I_Contact( #ConfigFB.Inicio_E1E3 )
   END_RUNG wire#w3
   RUNG wire#w2
      Contact( #Selec_M1_Salida )
      I_Contact( #ConfigFB.Final_E1E3 )
   END_RUNG wire#w3
   RUNG wire#powerrail
      Contact( #Mx_ET60 )
      wire#w4
      Contact( #Selec_M4_Salida )
      Contact( #AVTF_Ent_M2 )
      I_Contact( #ConfigFB.NoEntrar_E2 )
      Contact( #ConfigFB.Simultaneo_E2 )
      wire#w5
      I_Contact( #EstadoZona.ParoBlando_CBx )
      { S7_Templates := "SrcType := Int" } LE_Contact(in1 := #CNT_Simultaneo.CVD, in2 := #V_InicioSimultaneo)
      { S7_Templates := "SrcType := Int" } LE_Contact(in1 := #V_FinSimultaneo, in2 := #CNT_Simultaneo.CVD)
   END_RUNG wire#w3
   RUNG wire#powerrail
      Contact( #Mx_ET61 )
   END_RUNG wire#w4
   RUNG wire#w4
      Contact( #Selec_M2_Salida )
      Contact( #AVTF_Ent_M4 )
      I_Contact( #ConfigFB.NoEntrar_E4 )
      Contact( #ConfigFB.Simultaneo_E4 )
   END_RUNG wire#w5
   RUNG wire#w5
      Contact( #Selec_M4_Salida )
      I_Contact( #ConfigFB.Inicio_E2E4 )
   END_RUNG wire#w3
   RUNG wire#w5
      Contact( #Selec_M2_Salida )
      I_Contact( #ConfigFB.Final_E2E4 )
   END_RUNG wire#w3
   RUNG wire#powerrail
      I_Contact( #Mx_ET50 )
      I_Contact( #Mx_ET51 )
      I_Contact( #Mx_ET60 )
      I_Contact( #Mx_ET61 )
   END_RUNG wire#w6
   // the same network as SCL:
   IF (((#Mx_ET50 OR #Mx_ET51) AND ((#Selec_M3_Salida AND #AVTF_Ent_M1 AND NOT #ConfigFB.NoEntrar_E1 AND #ConfigFB.Simultaneo_E1) OR (#Selec_M1_Salida AND #AVTF_Ent_M3 AND NOT #ConfigFB.NoEntrar_E3 AND #ConfigFB.Simultaneo_E3)) AND ((NOT #EstadoZona.ParoBlando_CBx AND (#CNT_Simultaneo.CVD <= #V_InicioSimultaneo) AND (#V_FinSimultaneo <= #CNT_Simultaneo.CVD)) OR (#Selec_M3_Salida AND NOT #ConfigFB.Inicio_E1E3) OR (#Selec_M1_Salida AND NOT #ConfigFB.Final_E1E3))) OR ((#Mx_ET60 OR #Mx_ET61) AND ((#Selec_M4_Salida AND #AVTF_Ent_M2 AND NOT #ConfigFB.NoEntrar_E2 AND #ConfigFB.Simultaneo_E2) OR (#Selec_M2_Salida AND #AVTF_Ent_M4 AND NOT #ConfigFB.NoEntrar_E4 AND #ConfigFB.Simultaneo_E4)) AND ((NOT #EstadoZona.ParoBlando_CBx AND (#CNT_Simultaneo.CVD <= #V_InicioSimultaneo) AND (#V_FinSimultaneo <= #CNT_Simultaneo.CVD)) OR (#Selec_M4_Salida AND NOT #ConfigFB.Inicio_E2E4) OR (#Selec_M2_Salida AND NOT #ConfigFB.Final_E2E4)))) AND "ON" THEN
       #Simultaneo_Mx := TRUE;   // SR flip-flop
   END_IF;
   IF NOT #Mx_ET50 AND NOT #Mx_ET51 AND NOT #Mx_ET60 AND NOT #Mx_ET61 THEN #Simultaneo_Mx := FALSE; END_IF;
END_REGION

REGION Network 118: MENSAJES - PRESENCIA
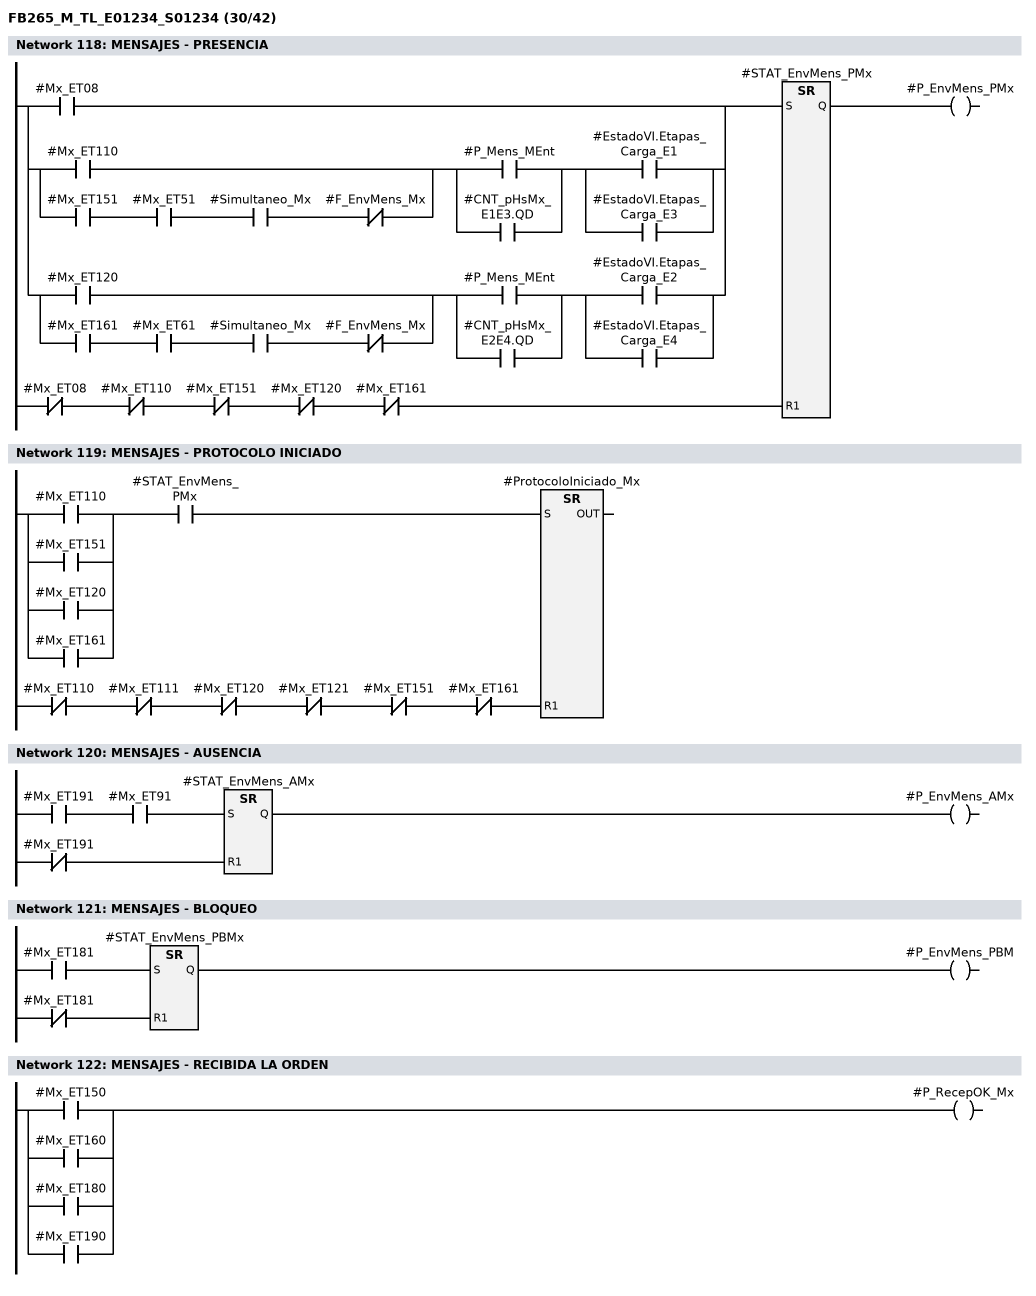
   RUNG wire#powerrail
      Contact( #Mx_ET08 )
      wire#w1
      S_SR(operand := #STAT_EnvMens_PMx, r1 := wire#w6)
      Coil( #P_EnvMens_PMx )
   END_RUNG
   RUNG wire#powerrail
      Contact( #Mx_ET110 )
      wire#w2
      Contact( #P_Mens_MEnt )
      wire#w3
      Contact( #EstadoVI.Etapas_Carga_E1 )
   END_RUNG wire#w1
   RUNG wire#powerrail
      Contact( #Mx_ET151 )
      Contact( #Mx_ET51 )
      Contact( #Simultaneo_Mx )
      I_Contact( #F_EnvMens_Mx )
   END_RUNG wire#w2
   RUNG wire#w2
      Contact( #CNT_pHsMx_E1E3.QD )
   END_RUNG wire#w3
   RUNG wire#w3
      Contact( #EstadoVI.Etapas_Carga_E3 )
   END_RUNG wire#w1
   RUNG wire#powerrail
      Contact( #Mx_ET120 )
      wire#w4
      Contact( #P_Mens_MEnt )
      wire#w5
      Contact( #EstadoVI.Etapas_Carga_E2 )
   END_RUNG wire#w1
   RUNG wire#powerrail
      Contact( #Mx_ET161 )
      Contact( #Mx_ET61 )
      Contact( #Simultaneo_Mx )
      I_Contact( #F_EnvMens_Mx )
   END_RUNG wire#w4
   RUNG wire#w4
      Contact( #CNT_pHsMx_E2E4.QD )
   END_RUNG wire#w5
   RUNG wire#w5
      Contact( #EstadoVI.Etapas_Carga_E4 )
   END_RUNG wire#w1
   RUNG wire#powerrail
      I_Contact( #Mx_ET08 )
      I_Contact( #Mx_ET110 )
      I_Contact( #Mx_ET151 )
      I_Contact( #Mx_ET120 )
      I_Contact( #Mx_ET161 )
   END_RUNG wire#w6
   // the same network as SCL:
   IF #Mx_ET08 OR ((#Mx_ET110 OR (#Mx_ET151 AND #Mx_ET51 AND #Simultaneo_Mx AND NOT #F_EnvMens_Mx)) AND (#P_Mens_MEnt OR #CNT_pHsMx_E1E3.QD) AND (#EstadoVI.Etapas_Carga_E1 OR #EstadoVI.Etapas_Carga_E3)) OR ((#Mx_ET120 OR (#Mx_ET161 AND #Mx_ET61 AND #Simultaneo_Mx AND NOT #F_EnvMens_Mx)) AND (#P_Mens_MEnt OR #CNT_pHsMx_E2E4.QD) AND (#EstadoVI.Etapas_Carga_E2 OR #EstadoVI.Etapas_Carga_E4)) THEN
       #STAT_EnvMens_PMx := TRUE;   // SR flip-flop
   END_IF;
   IF NOT #Mx_ET08 AND NOT #Mx_ET110 AND NOT #Mx_ET151 AND NOT #Mx_ET120 AND NOT #Mx_ET161 THEN
       #STAT_EnvMens_PMx := FALSE;
   END_IF;
   #P_EnvMens_PMx := #STAT_EnvMens_PMx;
END_REGION

REGION Network 119: MENSAJES - PROTOCOLO INICIADO
   RUNG wire#powerrail
      Contact( #Mx_ET110 )
      wire#w1
      Contact( #STAT_EnvMens_PMx )
      S_SR(operand := #ProtocoloIniciado_Mx, r1 := wire#w2)
   END_RUNG
   RUNG wire#powerrail
      Contact( #Mx_ET151 )
   END_RUNG wire#w1
   RUNG wire#powerrail
      Contact( #Mx_ET120 )
   END_RUNG wire#w1
   RUNG wire#powerrail
      Contact( #Mx_ET161 )
   END_RUNG wire#w1
   RUNG wire#powerrail
      I_Contact( #Mx_ET110 )
      I_Contact( #Mx_ET111 )
      I_Contact( #Mx_ET120 )
      I_Contact( #Mx_ET121 )
      I_Contact( #Mx_ET151 )
      I_Contact( #Mx_ET161 )
   END_RUNG wire#w2
   // the same network as SCL:
   IF (#Mx_ET110 OR #Mx_ET151 OR #Mx_ET120 OR #Mx_ET161) AND #STAT_EnvMens_PMx THEN
       #ProtocoloIniciado_Mx := TRUE;   // SR flip-flop
   END_IF;
   IF NOT #Mx_ET110 AND NOT #Mx_ET111 AND NOT #Mx_ET120 AND NOT #Mx_ET121 AND NOT #Mx_ET151 AND NOT #Mx_ET161 THEN
       #ProtocoloIniciado_Mx := FALSE;
   END_IF;
END_REGION

REGION Network 120: MENSAJES - AUSENCIA
   RUNG wire#powerrail
      Contact( #Mx_ET191 )
      Contact( #Mx_ET91 )
      S_SR(operand := #STAT_EnvMens_AMx, r1 := wire#w1)
      Coil( #P_EnvMens_AMx )
   END_RUNG
   RUNG wire#powerrail
      I_Contact( #Mx_ET191 )
   END_RUNG wire#w1
   // the same network as SCL:
   IF #Mx_ET191 AND #Mx_ET91 THEN
       #STAT_EnvMens_AMx := TRUE;   // SR flip-flop
   END_IF;
   IF NOT #Mx_ET191 THEN #STAT_EnvMens_AMx := FALSE; END_IF;
   #P_EnvMens_AMx := #STAT_EnvMens_AMx;
END_REGION

REGION Network 121: MENSAJES - BLOQUEO
   RUNG wire#powerrail
      Contact( #Mx_ET181 )
      S_SR(operand := #STAT_EnvMens_PBMx, r1 := wire#w1)
      Coil( #P_EnvMens_PBM )
   END_RUNG
   RUNG wire#powerrail
      I_Contact( #Mx_ET181 )
   END_RUNG wire#w1
   // the same network as SCL:
   IF #Mx_ET181 THEN
       #STAT_EnvMens_PBMx := TRUE;   // SR flip-flop
   END_IF;
   IF NOT #Mx_ET181 THEN #STAT_EnvMens_PBMx := FALSE; END_IF;
   #P_EnvMens_PBM := #STAT_EnvMens_PBMx;
END_REGION

REGION Network 122: MENSAJES - RECIBIDA LA ORDEN
   RUNG wire#powerrail
      Contact( #Mx_ET150 )
      wire#w1
      Coil( #P_RecepOK_Mx )
   END_RUNG
   RUNG wire#powerrail
      Contact( #Mx_ET160 )
   END_RUNG wire#w1
   RUNG wire#powerrail
      Contact( #Mx_ET180 )
   END_RUNG wire#w1
   RUNG wire#powerrail
      Contact( #Mx_ET190 )
   END_RUNG wire#w1
   // the same network as SCL:
   #P_RecepOK_Mx := #Mx_ET150 OR #Mx_ET160 OR #Mx_ET180 OR #Mx_ET190;
END_REGION

REGION Network 123: VARIABLES AUXILIARES - OK TP01 ABAJO
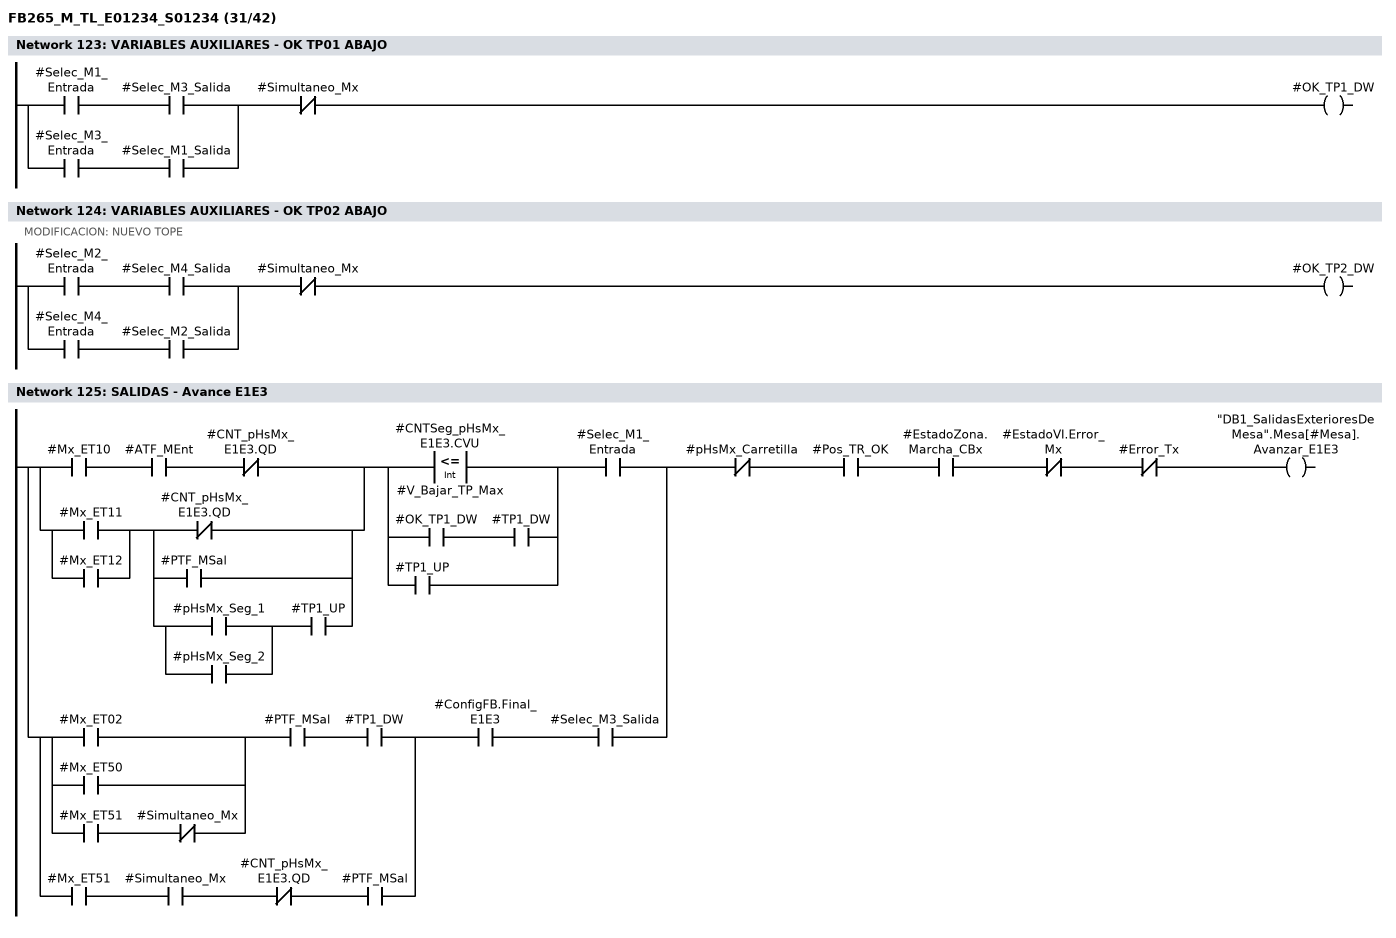
   RUNG wire#powerrail
      Contact( #Selec_M1_Entrada )
      Contact( #Selec_M3_Salida )
      wire#w1
      I_Contact( #Simultaneo_Mx )
      Coil( #OK_TP1_DW )
   END_RUNG
   RUNG wire#powerrail
      Contact( #Selec_M3_Entrada )
      Contact( #Selec_M1_Salida )
   END_RUNG wire#w1
   // the same network as SCL:
   #OK_TP1_DW := ((#Selec_M1_Entrada AND #Selec_M3_Salida) OR (#Selec_M3_Entrada AND #Selec_M1_Salida)) AND NOT #Simultaneo_Mx;
END_REGION

REGION Network 124: VARIABLES AUXILIARES - OK TP02 ABAJO
   // MODIFICACION: NUEVO TOPE
   RUNG wire#powerrail
      Contact( #Selec_M2_Entrada )
      Contact( #Selec_M4_Salida )
      wire#w1
      I_Contact( #Simultaneo_Mx )
      Coil( #OK_TP2_DW )
   END_RUNG
   RUNG wire#powerrail
      Contact( #Selec_M4_Entrada )
      Contact( #Selec_M2_Salida )
   END_RUNG wire#w1
   // the same network as SCL:
   #OK_TP2_DW := ((#Selec_M2_Entrada AND #Selec_M4_Salida) OR (#Selec_M4_Entrada AND #Selec_M2_Salida)) AND NOT #Simultaneo_Mx;
END_REGION

REGION Network 125: SALIDAS - Avance E1E3
   RUNG wire#powerrail
      Contact( #Mx_ET10 )
      Contact( #ATF_MEnt )
      I_Contact( #CNT_pHsMx_E1E3.QD )
      wire#w1
      { S7_Templates := "SrcType := Int" } LE_Contact(in1 := #CNTSeg_pHsMx_E1E3.CVU, in2 := #V_Bajar_TP_Max)
      wire#w4
      Contact( #Selec_M1_Entrada )
      wire#w5
      I_Contact( #pHsMx_Carretilla )
      Contact( #Pos_TR_OK )
      Contact( #EstadoZona.Marcha_CBx )
      I_Contact( #EstadoVI.Error_Mx )
      I_Contact( #Error_Tx )
      Coil( "DB1_SalidasExterioresDeMesa".Mesa[#Mesa].Avanzar_E1E3 )
   END_RUNG
   RUNG wire#powerrail
      Contact( #Mx_ET11 )
      wire#w2
      I_Contact( #CNT_pHsMx_E1E3.QD )
   END_RUNG wire#w1
   RUNG wire#powerrail
      Contact( #Mx_ET12 )
   END_RUNG wire#w2
   RUNG wire#w2
      Contact( #PTF_MSal )
   END_RUNG wire#w1
   RUNG wire#w2
      Contact( #pHsMx_Seg_1 )
      wire#w3
      Contact( #TP1_UP )
   END_RUNG wire#w1
   RUNG wire#w2
      Contact( #pHsMx_Seg_2 )
   END_RUNG wire#w3
   RUNG wire#w1
      Contact( #OK_TP1_DW )
      Contact( #TP1_DW )
   END_RUNG wire#w4
   RUNG wire#w1
      Contact( #TP1_UP )
   END_RUNG wire#w4
   RUNG wire#powerrail
      Contact( #Mx_ET02 )
      wire#w6
      Contact( #PTF_MSal )
      Contact( #TP1_DW )
      wire#w7
      Contact( #ConfigFB.Final_E1E3 )
      Contact( #Selec_M3_Salida )
   END_RUNG wire#w5
   RUNG wire#powerrail
      Contact( #Mx_ET50 )
   END_RUNG wire#w6
   RUNG wire#powerrail
      Contact( #Mx_ET51 )
      I_Contact( #Simultaneo_Mx )
   END_RUNG wire#w6
   RUNG wire#powerrail
      Contact( #Mx_ET51 )
      Contact( #Simultaneo_Mx )
      I_Contact( #CNT_pHsMx_E1E3.QD )
      Contact( #PTF_MSal )
   END_RUNG wire#w7
   // the same network as SCL:
   "DB1_SalidasExterioresDeMesa".Mesa[#Mesa].Avanzar_E1E3 := ((((#Mx_ET10 AND #ATF_MEnt AND NOT #CNT_pHsMx_E1E3.QD) OR ((#Mx_ET11 OR #Mx_ET12) AND (NOT #CNT_pHsMx_E1E3.QD OR #PTF_MSal OR ((#pHsMx_Seg_1 OR #pHsMx_Seg_2) AND #TP1_UP)))) AND ((#CNTSeg_pHsMx_E1E3.CVU <= #V_Bajar_TP_Max) OR (#OK_TP1_DW AND #TP1_DW) OR #TP1_UP) AND #Selec_M1_Entrada) OR ((((#Mx_ET02 OR #Mx_ET50 OR (#Mx_ET51 AND NOT #Simultaneo_Mx)) AND #PTF_MSal AND #TP1_DW) OR (#Mx_ET51 AND #Simultaneo_Mx AND NOT #CNT_pHsMx_E1E3.QD AND #PTF_MSal)) AND #ConfigFB.Final_E1E3 AND #Selec_M3_Salida)) AND NOT #pHsMx_Carretilla AND #Pos_TR_OK AND #EstadoZona.Marcha_CBx AND NOT #EstadoVI.Error_Mx AND NOT #Error_Tx;
END_REGION

REGION Network 126: SALIDAS - Retroceso E1E3
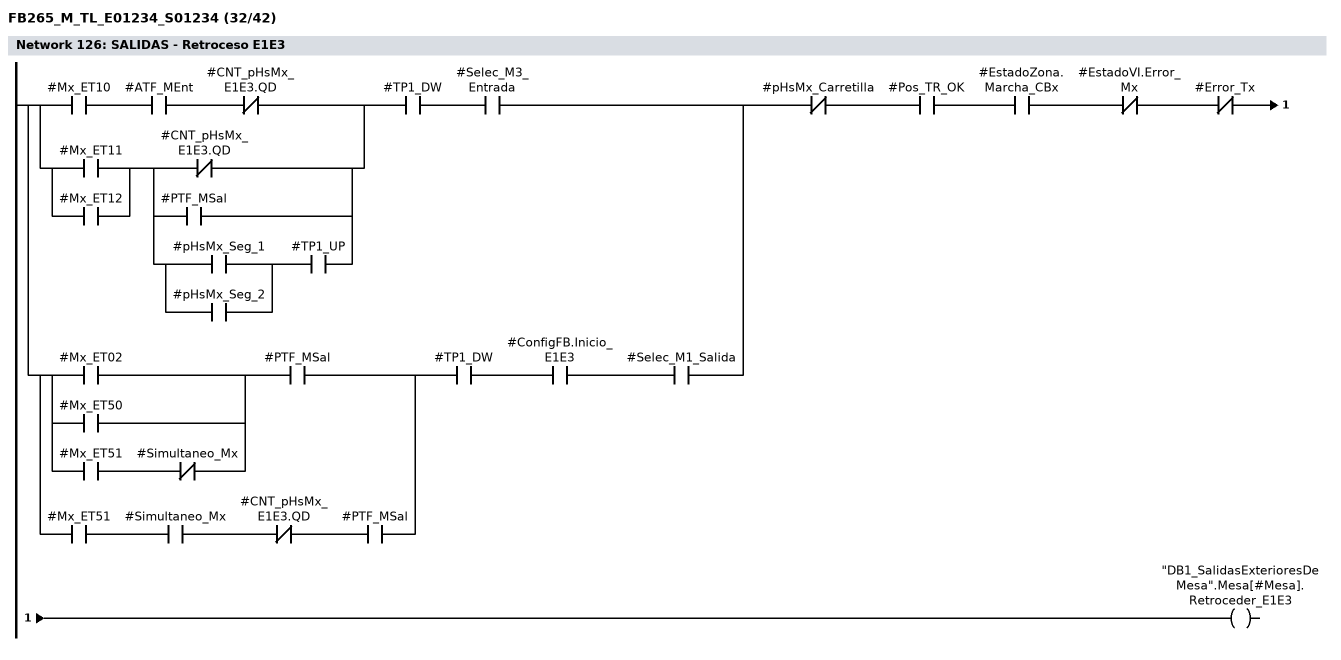
   RUNG wire#powerrail
      Contact( #Mx_ET10 )
      Contact( #ATF_MEnt )
      I_Contact( #CNT_pHsMx_E1E3.QD )
      wire#w1
      Contact( #TP1_DW )
      Contact( #Selec_M3_Entrada )
      wire#w4
      I_Contact( #pHsMx_Carretilla )
      Contact( #Pos_TR_OK )
      Contact( #EstadoZona.Marcha_CBx )
      I_Contact( #EstadoVI.Error_Mx )
      I_Contact( #Error_Tx )
      Coil( "DB1_SalidasExterioresDeMesa".Mesa[#Mesa].Retroceder_E1E3 )
   END_RUNG
   RUNG wire#powerrail
      Contact( #Mx_ET11 )
      wire#w2
      I_Contact( #CNT_pHsMx_E1E3.QD )
   END_RUNG wire#w1
   RUNG wire#powerrail
      Contact( #Mx_ET12 )
   END_RUNG wire#w2
   RUNG wire#w2
      Contact( #PTF_MSal )
   END_RUNG wire#w1
   RUNG wire#w2
      Contact( #pHsMx_Seg_1 )
      wire#w3
      Contact( #TP1_UP )
   END_RUNG wire#w1
   RUNG wire#w2
      Contact( #pHsMx_Seg_2 )
   END_RUNG wire#w3
   RUNG wire#powerrail
      Contact( #Mx_ET02 )
      wire#w5
      Contact( #PTF_MSal )
      wire#w6
      Contact( #TP1_DW )
      Contact( #ConfigFB.Inicio_E1E3 )
      Contact( #Selec_M1_Salida )
   END_RUNG wire#w4
   RUNG wire#powerrail
      Contact( #Mx_ET50 )
   END_RUNG wire#w5
   RUNG wire#powerrail
      Contact( #Mx_ET51 )
      I_Contact( #Simultaneo_Mx )
   END_RUNG wire#w5
   RUNG wire#powerrail
      Contact( #Mx_ET51 )
      Contact( #Simultaneo_Mx )
      I_Contact( #CNT_pHsMx_E1E3.QD )
      Contact( #PTF_MSal )
   END_RUNG wire#w6
   // the same network as SCL:
   "DB1_SalidasExterioresDeMesa".Mesa[#Mesa].Retroceder_E1E3 := ((((#Mx_ET10 AND #ATF_MEnt AND NOT #CNT_pHsMx_E1E3.QD) OR ((#Mx_ET11 OR #Mx_ET12) AND (NOT #CNT_pHsMx_E1E3.QD OR #PTF_MSal OR ((#pHsMx_Seg_1 OR #pHsMx_Seg_2) AND #TP1_UP)))) AND #TP1_DW AND #Selec_M3_Entrada) OR ((((#Mx_ET02 OR #Mx_ET50 OR (#Mx_ET51 AND NOT #Simultaneo_Mx)) AND #PTF_MSal) OR (#Mx_ET51 AND #Simultaneo_Mx AND NOT #CNT_pHsMx_E1E3.QD AND #PTF_MSal)) AND #TP1_DW AND #ConfigFB.Inicio_E1E3 AND #Selec_M1_Salida)) AND NOT #pHsMx_Carretilla AND #Pos_TR_OK AND #EstadoZona.Marcha_CBx AND NOT #EstadoVI.Error_Mx AND NOT #Error_Tx;
END_REGION

REGION Network 127: SALIDAS - Parar E1E3
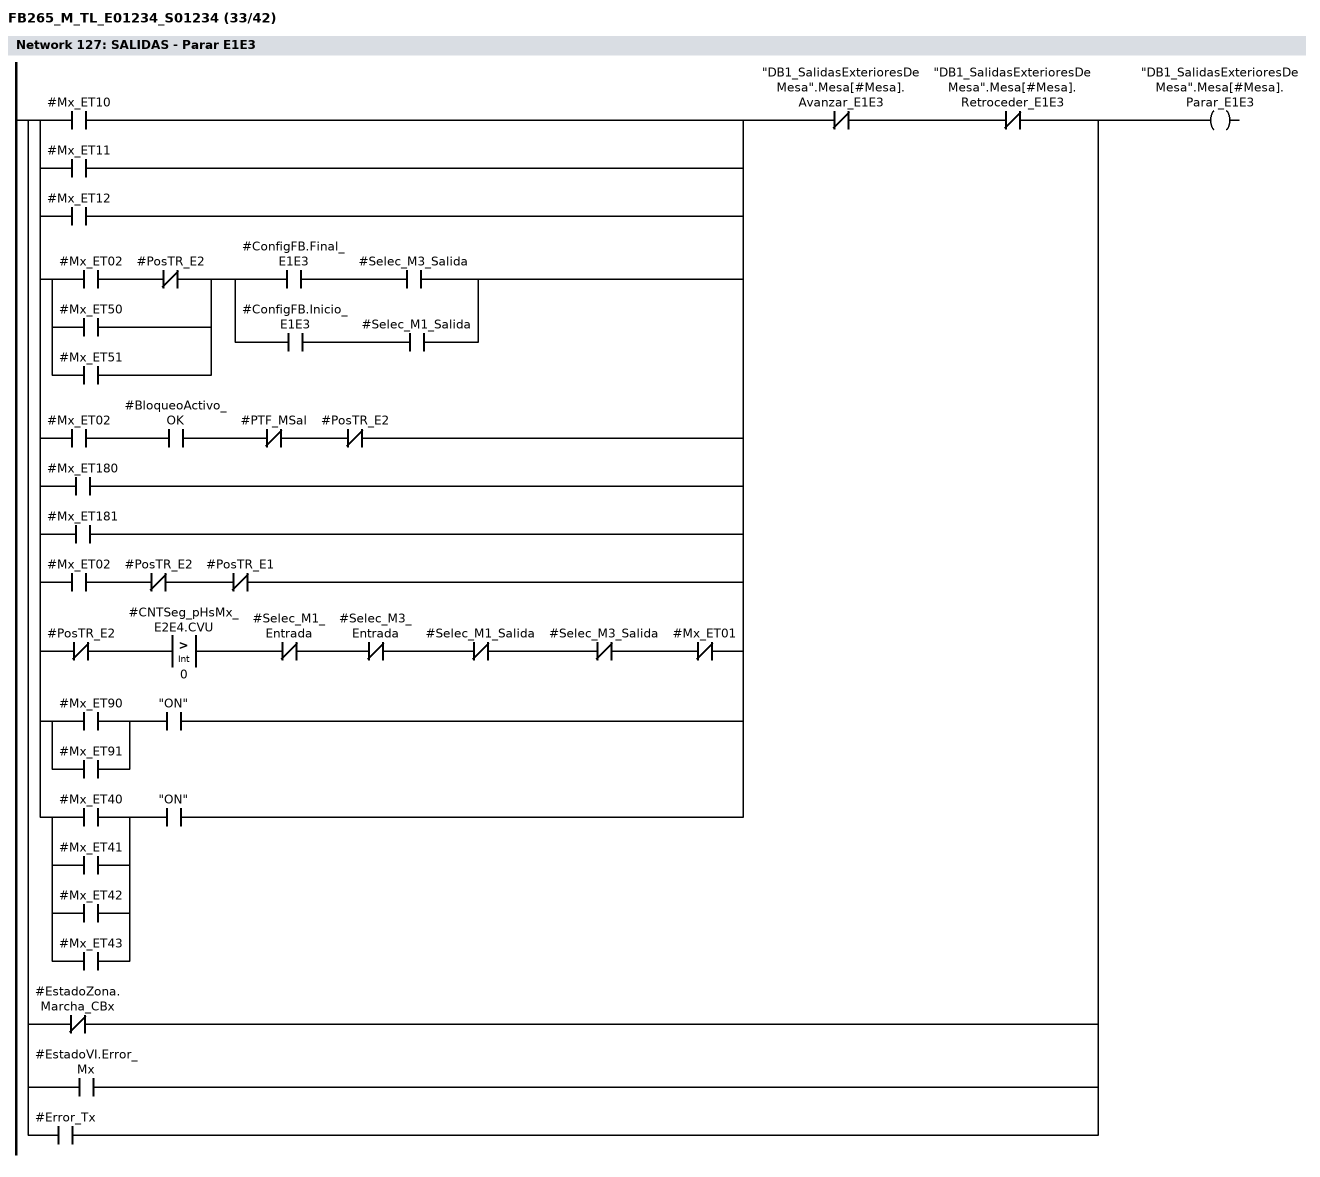
   RUNG wire#powerrail
      Contact( #Mx_ET10 )
      wire#w1
      I_Contact( "DB1_SalidasExterioresDeMesa".Mesa[#Mesa].Avanzar_E1E3 )
      I_Contact( "DB1_SalidasExterioresDeMesa".Mesa[#Mesa].Retroceder_E1E3 )
      wire#w5
      Coil( "DB1_SalidasExterioresDeMesa".Mesa[#Mesa].Parar_E1E3 )
   END_RUNG
   RUNG wire#powerrail
      Contact( #Mx_ET11 )
   END_RUNG wire#w1
   RUNG wire#powerrail
      Contact( #Mx_ET12 )
   END_RUNG wire#w1
   RUNG wire#powerrail
      Contact( #Mx_ET02 )
      I_Contact( #PosTR_E2 )
      wire#w2
      Contact( #ConfigFB.Final_E1E3 )
      Contact( #Selec_M3_Salida )
   END_RUNG wire#w1
   RUNG wire#powerrail
      Contact( #Mx_ET50 )
   END_RUNG wire#w2
   RUNG wire#powerrail
      Contact( #Mx_ET51 )
   END_RUNG wire#w2
   RUNG wire#w2
      Contact( #ConfigFB.Inicio_E1E3 )
      Contact( #Selec_M1_Salida )
   END_RUNG wire#w1
   RUNG wire#powerrail
      Contact( #Mx_ET02 )
      Contact( #BloqueoActivo_OK )
      I_Contact( #PTF_MSal )
      I_Contact( #PosTR_E2 )
   END_RUNG wire#w1
   RUNG wire#powerrail
      Contact( #Mx_ET180 )
   END_RUNG wire#w1
   RUNG wire#powerrail
      Contact( #Mx_ET181 )
   END_RUNG wire#w1
   RUNG wire#powerrail
      Contact( #Mx_ET02 )
      I_Contact( #PosTR_E2 )
      I_Contact( #PosTR_E1 )
   END_RUNG wire#w1
   RUNG wire#powerrail
      I_Contact( #PosTR_E2 )
      { S7_Templates := "SrcType := Int" } GT_Contact(in1 := #CNTSeg_pHsMx_E2E4.CVU, in2 := 0)
      I_Contact( #Selec_M1_Entrada )
      I_Contact( #Selec_M3_Entrada )
      I_Contact( #Selec_M1_Salida )
      I_Contact( #Selec_M3_Salida )
      I_Contact( #Mx_ET01 )
   END_RUNG wire#w1
   RUNG wire#powerrail
      Contact( #Mx_ET90 )
      wire#w3
      Contact( "ON" )
   END_RUNG wire#w1
   RUNG wire#powerrail
      Contact( #Mx_ET91 )
   END_RUNG wire#w3
   RUNG wire#powerrail
      Contact( #Mx_ET40 )
      wire#w4
      Contact( "ON" )
   END_RUNG wire#w1
   RUNG wire#powerrail
      Contact( #Mx_ET41 )
   END_RUNG wire#w4
   RUNG wire#powerrail
      Contact( #Mx_ET42 )
   END_RUNG wire#w4
   RUNG wire#powerrail
      Contact( #Mx_ET43 )
   END_RUNG wire#w4
   RUNG wire#powerrail
      I_Contact( #EstadoZona.Marcha_CBx )
   END_RUNG wire#w5
   RUNG wire#powerrail
      Contact( #EstadoVI.Error_Mx )
   END_RUNG wire#w5
   RUNG wire#powerrail
      Contact( #Error_Tx )
   END_RUNG wire#w5
   // the same network as SCL:
   "DB1_SalidasExterioresDeMesa".Mesa[#Mesa].Parar_E1E3 := ((#Mx_ET10 OR #Mx_ET11 OR #Mx_ET12 OR (((#Mx_ET02 AND NOT #PosTR_E2) OR #Mx_ET50 OR #Mx_ET51) AND ((#ConfigFB.Final_E1E3 AND #Selec_M3_Salida) OR (#ConfigFB.Inicio_E1E3 AND #Selec_M1_Salida))) OR (#Mx_ET02 AND #BloqueoActivo_OK AND NOT #PTF_MSal AND NOT #PosTR_E2) OR #Mx_ET180 OR #Mx_ET181 OR (#Mx_ET02 AND NOT #PosTR_E2 AND NOT #PosTR_E1) OR (NOT #PosTR_E2 AND (#CNTSeg_pHsMx_E2E4.CVU > 0) AND NOT #Selec_M1_Entrada AND NOT #Selec_M3_Entrada AND NOT #Selec_M1_Salida AND NOT #Selec_M3_Salida AND NOT #Mx_ET01) OR ((#Mx_ET90 OR #Mx_ET91) AND "ON") OR ((#Mx_ET40 OR #Mx_ET41 OR #Mx_ET42 OR #Mx_ET43) AND "ON")) AND NOT "DB1_SalidasExterioresDeMesa".Mesa[#Mesa].Avanzar_E1E3 AND NOT "DB1_SalidasExterioresDeMesa".Mesa[#Mesa].Retroceder_E1E3) OR NOT #EstadoZona.Marcha_CBx OR #EstadoVI.Error_Mx OR #Error_Tx;
END_REGION

REGION Network 128: SALIDAS - Valor Frecuencia Lenta E1E3
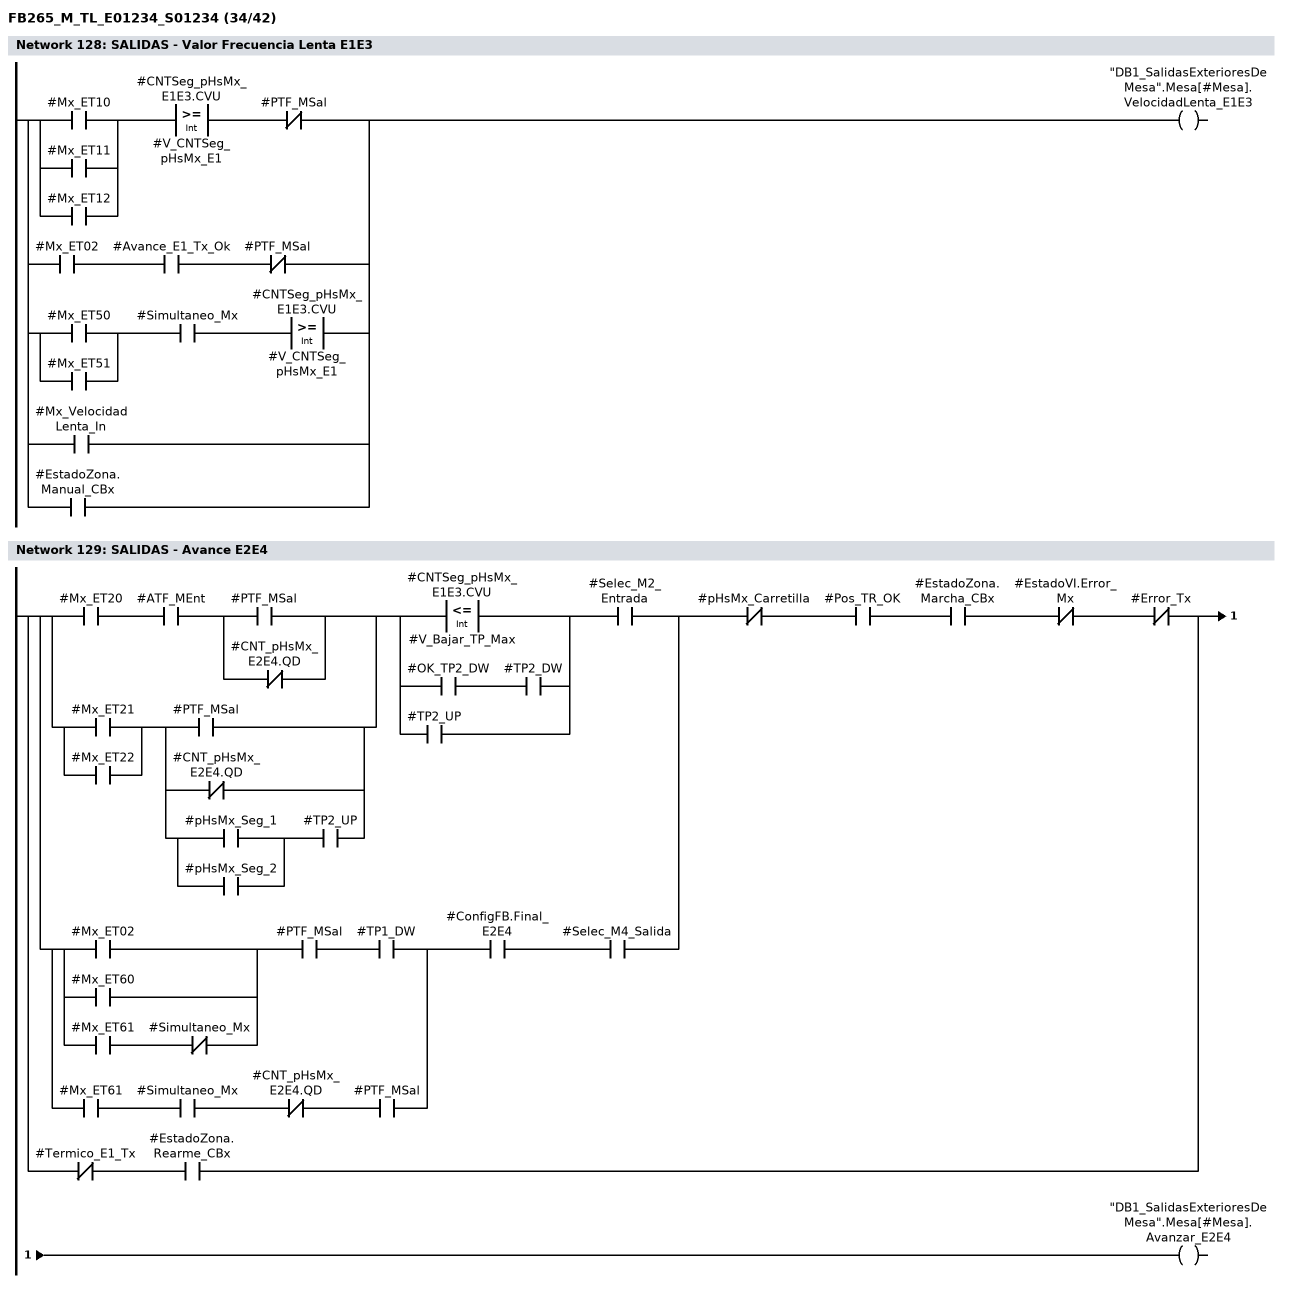
   RUNG wire#powerrail
      Contact( #Mx_ET10 )
      wire#w1
      { S7_Templates := "SrcType := Int" } GE_Contact(in1 := #CNTSeg_pHsMx_E1E3.CVU, in2 := #V_CNTSeg_pHsMx_E1)
      I_Contact( #PTF_MSal )
      wire#w2
      Coil( "DB1_SalidasExterioresDeMesa".Mesa[#Mesa].VelocidadLenta_E1E3 )
   END_RUNG
   RUNG wire#powerrail
      Contact( #Mx_ET11 )
   END_RUNG wire#w1
   RUNG wire#powerrail
      Contact( #Mx_ET12 )
   END_RUNG wire#w1
   RUNG wire#powerrail
      Contact( #Mx_ET02 )
      Contact( #Avance_E1_Tx_Ok )
      I_Contact( #PTF_MSal )
   END_RUNG wire#w2
   RUNG wire#powerrail
      Contact( #Mx_ET50 )
      wire#w3
      Contact( #Simultaneo_Mx )
      { S7_Templates := "SrcType := Int" } GE_Contact(in1 := #CNTSeg_pHsMx_E1E3.CVU, in2 := #V_CNTSeg_pHsMx_E1)
   END_RUNG wire#w2
   RUNG wire#powerrail
      Contact( #Mx_ET51 )
   END_RUNG wire#w3
   RUNG wire#powerrail
      Contact( #Mx_VelocidadLenta_In )
   END_RUNG wire#w2
   RUNG wire#powerrail
      Contact( #EstadoZona.Manual_CBx )
   END_RUNG wire#w2
   // the same network as SCL:
   "DB1_SalidasExterioresDeMesa".Mesa[#Mesa].VelocidadLenta_E1E3 := ((#Mx_ET10 OR #Mx_ET11 OR #Mx_ET12) AND (#CNTSeg_pHsMx_E1E3.CVU >= #V_CNTSeg_pHsMx_E1) AND NOT #PTF_MSal) OR (#Mx_ET02 AND #Avance_E1_Tx_Ok AND NOT #PTF_MSal) OR ((#Mx_ET50 OR #Mx_ET51) AND #Simultaneo_Mx AND (#CNTSeg_pHsMx_E1E3.CVU >= #V_CNTSeg_pHsMx_E1)) OR #Mx_VelocidadLenta_In OR #EstadoZona.Manual_CBx;
END_REGION

REGION Network 129: SALIDAS - Avance E2E4
   RUNG wire#powerrail
      Contact( #Mx_ET20 )
      Contact( #ATF_MEnt )
      wire#w1
      Contact( #PTF_MSal )
      wire#w2
      { S7_Templates := "SrcType := Int" } LE_Contact(in1 := #CNTSeg_pHsMx_E1E3.CVU, in2 := #V_Bajar_TP_Max)
      wire#w5
      Contact( #Selec_M2_Entrada )
      wire#w6
      I_Contact( #pHsMx_Carretilla )
      Contact( #Pos_TR_OK )
      Contact( #EstadoZona.Marcha_CBx )
      I_Contact( #EstadoVI.Error_Mx )
      I_Contact( #Error_Tx )
      wire#w9
      Coil( "DB1_SalidasExterioresDeMesa".Mesa[#Mesa].Avanzar_E2E4 )
   END_RUNG
   RUNG wire#w1
      I_Contact( #CNT_pHsMx_E2E4.QD )
   END_RUNG wire#w2
   RUNG wire#powerrail
      Contact( #Mx_ET21 )
      wire#w3
      Contact( #PTF_MSal )
   END_RUNG wire#w2
   RUNG wire#powerrail
      Contact( #Mx_ET22 )
   END_RUNG wire#w3
   RUNG wire#w3
      I_Contact( #CNT_pHsMx_E2E4.QD )
   END_RUNG wire#w2
   RUNG wire#w3
      Contact( #pHsMx_Seg_1 )
      wire#w4
      Contact( #TP2_UP )
   END_RUNG wire#w2
   RUNG wire#w3
      Contact( #pHsMx_Seg_2 )
   END_RUNG wire#w4
   RUNG wire#w2
      Contact( #OK_TP2_DW )
      Contact( #TP2_DW )
   END_RUNG wire#w5
   RUNG wire#w2
      Contact( #TP2_UP )
   END_RUNG wire#w5
   RUNG wire#powerrail
      Contact( #Mx_ET02 )
      wire#w7
      Contact( #PTF_MSal )
      Contact( #TP1_DW )
      wire#w8
      Contact( #ConfigFB.Final_E2E4 )
      Contact( #Selec_M4_Salida )
   END_RUNG wire#w6
   RUNG wire#powerrail
      Contact( #Mx_ET60 )
   END_RUNG wire#w7
   RUNG wire#powerrail
      Contact( #Mx_ET61 )
      I_Contact( #Simultaneo_Mx )
   END_RUNG wire#w7
   RUNG wire#powerrail
      Contact( #Mx_ET61 )
      Contact( #Simultaneo_Mx )
      I_Contact( #CNT_pHsMx_E2E4.QD )
      Contact( #PTF_MSal )
   END_RUNG wire#w8
   RUNG wire#powerrail
      I_Contact( #Termico_E1_Tx )
      Contact( #EstadoZona.Rearme_CBx )
   END_RUNG wire#w9
   // the same network as SCL:
   "DB1_SalidasExterioresDeMesa".Mesa[#Mesa].Avanzar_E2E4 := (((((#Mx_ET20 AND #ATF_MEnt AND (#PTF_MSal OR NOT #CNT_pHsMx_E2E4.QD)) OR ((#Mx_ET21 OR #Mx_ET22) AND (#PTF_MSal OR NOT #CNT_pHsMx_E2E4.QD OR ((#pHsMx_Seg_1 OR #pHsMx_Seg_2) AND #TP2_UP)))) AND ((#CNTSeg_pHsMx_E1E3.CVU <= #V_Bajar_TP_Max) OR (#OK_TP2_DW AND #TP2_DW) OR #TP2_UP) AND #Selec_M2_Entrada) OR ((((#Mx_ET02 OR #Mx_ET60 OR (#Mx_ET61 AND NOT #Simultaneo_Mx)) AND #PTF_MSal AND #TP1_DW) OR (#Mx_ET61 AND #Simultaneo_Mx AND NOT #CNT_pHsMx_E2E4.QD AND #PTF_MSal)) AND #ConfigFB.Final_E2E4 AND #Selec_M4_Salida)) AND NOT #pHsMx_Carretilla AND #Pos_TR_OK AND #EstadoZona.Marcha_CBx AND NOT #EstadoVI.Error_Mx AND NOT #Error_Tx) OR (NOT #Termico_E1_Tx AND #EstadoZona.Rearme_CBx);
END_REGION

REGION Network 130: SALIDAS - Retroceso E2E4
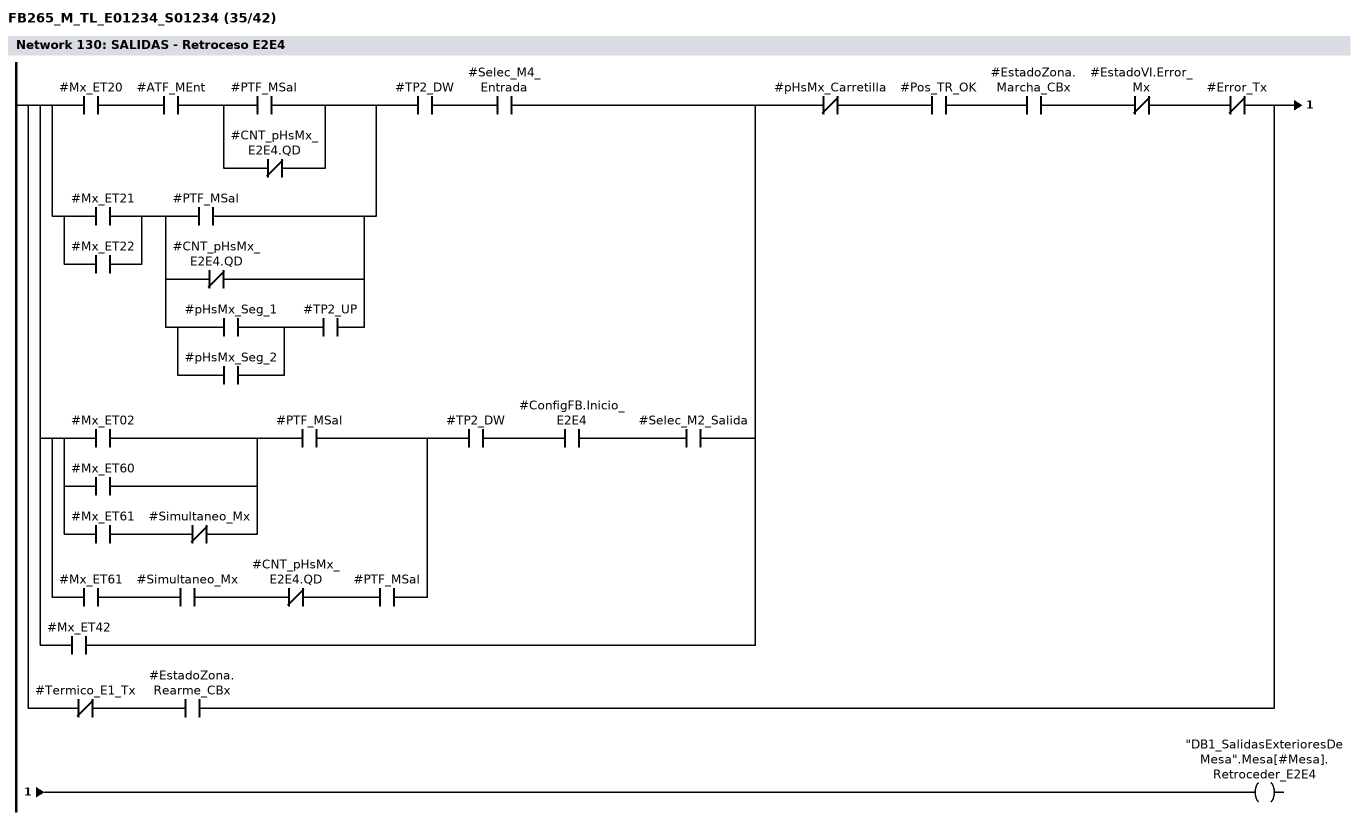
   RUNG wire#powerrail
      Contact( #Mx_ET20 )
      Contact( #ATF_MEnt )
      wire#w1
      Contact( #PTF_MSal )
      wire#w2
      Contact( #TP2_DW )
      Contact( #Selec_M4_Entrada )
      wire#w5
      I_Contact( #pHsMx_Carretilla )
      Contact( #Pos_TR_OK )
      Contact( #EstadoZona.Marcha_CBx )
      I_Contact( #EstadoVI.Error_Mx )
      I_Contact( #Error_Tx )
      wire#w8
      Coil( "DB1_SalidasExterioresDeMesa".Mesa[#Mesa].Retroceder_E2E4 )
   END_RUNG
   RUNG wire#w1
      I_Contact( #CNT_pHsMx_E2E4.QD )
   END_RUNG wire#w2
   RUNG wire#powerrail
      Contact( #Mx_ET21 )
      wire#w3
      Contact( #PTF_MSal )
   END_RUNG wire#w2
   RUNG wire#powerrail
      Contact( #Mx_ET22 )
   END_RUNG wire#w3
   RUNG wire#w3
      I_Contact( #CNT_pHsMx_E2E4.QD )
   END_RUNG wire#w2
   RUNG wire#w3
      Contact( #pHsMx_Seg_1 )
      wire#w4
      Contact( #TP2_UP )
   END_RUNG wire#w2
   RUNG wire#w3
      Contact( #pHsMx_Seg_2 )
   END_RUNG wire#w4
   RUNG wire#powerrail
      Contact( #Mx_ET02 )
      wire#w6
      Contact( #PTF_MSal )
      wire#w7
      Contact( #TP2_DW )
      Contact( #ConfigFB.Inicio_E2E4 )
      Contact( #Selec_M2_Salida )
   END_RUNG wire#w5
   RUNG wire#powerrail
      Contact( #Mx_ET60 )
   END_RUNG wire#w6
   RUNG wire#powerrail
      Contact( #Mx_ET61 )
      I_Contact( #Simultaneo_Mx )
   END_RUNG wire#w6
   RUNG wire#powerrail
      Contact( #Mx_ET61 )
      Contact( #Simultaneo_Mx )
      I_Contact( #CNT_pHsMx_E2E4.QD )
      Contact( #PTF_MSal )
   END_RUNG wire#w7
   RUNG wire#powerrail
      Contact( #Mx_ET42 )
   END_RUNG wire#w5
   RUNG wire#powerrail
      I_Contact( #Termico_E1_Tx )
      Contact( #EstadoZona.Rearme_CBx )
   END_RUNG wire#w8
   // the same network as SCL:
   "DB1_SalidasExterioresDeMesa".Mesa[#Mesa].Retroceder_E2E4 := (((((#Mx_ET20 AND #ATF_MEnt AND (#PTF_MSal OR NOT #CNT_pHsMx_E2E4.QD)) OR ((#Mx_ET21 OR #Mx_ET22) AND (#PTF_MSal OR NOT #CNT_pHsMx_E2E4.QD OR ((#pHsMx_Seg_1 OR #pHsMx_Seg_2) AND #TP2_UP)))) AND #TP2_DW AND #Selec_M4_Entrada) OR ((((#Mx_ET02 OR #Mx_ET60 OR (#Mx_ET61 AND NOT #Simultaneo_Mx)) AND #PTF_MSal) OR (#Mx_ET61 AND #Simultaneo_Mx AND NOT #CNT_pHsMx_E2E4.QD AND #PTF_MSal)) AND #TP2_DW AND #ConfigFB.Inicio_E2E4 AND #Selec_M2_Salida) OR #Mx_ET42) AND NOT #pHsMx_Carretilla AND #Pos_TR_OK AND #EstadoZona.Marcha_CBx AND NOT #EstadoVI.Error_Mx AND NOT #Error_Tx) OR (NOT #Termico_E1_Tx AND #EstadoZona.Rearme_CBx);
END_REGION

REGION Network 131: SALIDAS - Parar E2E4
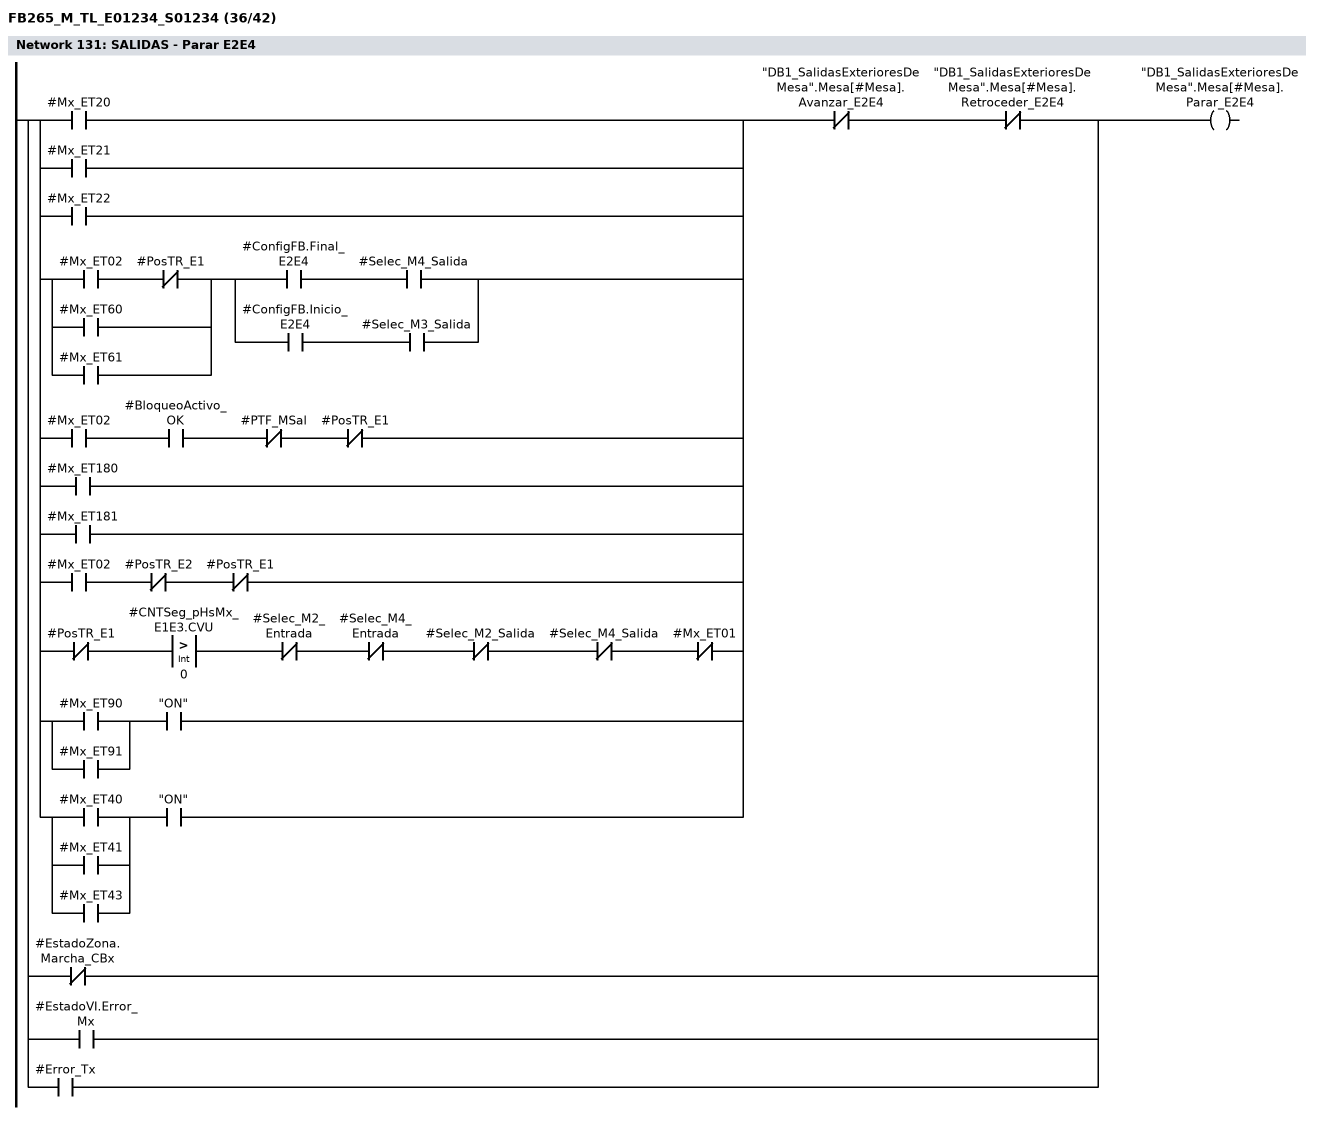
   RUNG wire#powerrail
      Contact( #Mx_ET20 )
      wire#w1
      I_Contact( "DB1_SalidasExterioresDeMesa".Mesa[#Mesa].Avanzar_E2E4 )
      I_Contact( "DB1_SalidasExterioresDeMesa".Mesa[#Mesa].Retroceder_E2E4 )
      wire#w5
      Coil( "DB1_SalidasExterioresDeMesa".Mesa[#Mesa].Parar_E2E4 )
   END_RUNG
   RUNG wire#powerrail
      Contact( #Mx_ET21 )
   END_RUNG wire#w1
   RUNG wire#powerrail
      Contact( #Mx_ET22 )
   END_RUNG wire#w1
   RUNG wire#powerrail
      Contact( #Mx_ET02 )
      I_Contact( #PosTR_E1 )
      wire#w2
      Contact( #ConfigFB.Final_E2E4 )
      Contact( #Selec_M4_Salida )
   END_RUNG wire#w1
   RUNG wire#powerrail
      Contact( #Mx_ET60 )
   END_RUNG wire#w2
   RUNG wire#powerrail
      Contact( #Mx_ET61 )
   END_RUNG wire#w2
   RUNG wire#w2
      Contact( #ConfigFB.Inicio_E2E4 )
      Contact( #Selec_M3_Salida )
   END_RUNG wire#w1
   RUNG wire#powerrail
      Contact( #Mx_ET02 )
      Contact( #BloqueoActivo_OK )
      I_Contact( #PTF_MSal )
      I_Contact( #PosTR_E1 )
   END_RUNG wire#w1
   RUNG wire#powerrail
      Contact( #Mx_ET180 )
   END_RUNG wire#w1
   RUNG wire#powerrail
      Contact( #Mx_ET181 )
   END_RUNG wire#w1
   RUNG wire#powerrail
      Contact( #Mx_ET02 )
      I_Contact( #PosTR_E2 )
      I_Contact( #PosTR_E1 )
   END_RUNG wire#w1
   RUNG wire#powerrail
      I_Contact( #PosTR_E1 )
      { S7_Templates := "SrcType := Int" } GT_Contact(in1 := #CNTSeg_pHsMx_E1E3.CVU, in2 := 0)
      I_Contact( #Selec_M2_Entrada )
      I_Contact( #Selec_M4_Entrada )
      I_Contact( #Selec_M2_Salida )
      I_Contact( #Selec_M4_Salida )
      I_Contact( #Mx_ET01 )
   END_RUNG wire#w1
   RUNG wire#powerrail
      Contact( #Mx_ET90 )
      wire#w3
      Contact( "ON" )
   END_RUNG wire#w1
   RUNG wire#powerrail
      Contact( #Mx_ET91 )
   END_RUNG wire#w3
   RUNG wire#powerrail
      Contact( #Mx_ET40 )
      wire#w4
      Contact( "ON" )
   END_RUNG wire#w1
   RUNG wire#powerrail
      Contact( #Mx_ET41 )
   END_RUNG wire#w4
   RUNG wire#powerrail
      Contact( #Mx_ET43 )
   END_RUNG wire#w4
   RUNG wire#powerrail
      I_Contact( #EstadoZona.Marcha_CBx )
   END_RUNG wire#w5
   RUNG wire#powerrail
      Contact( #EstadoVI.Error_Mx )
   END_RUNG wire#w5
   RUNG wire#powerrail
      Contact( #Error_Tx )
   END_RUNG wire#w5
   // the same network as SCL:
   "DB1_SalidasExterioresDeMesa".Mesa[#Mesa].Parar_E2E4 := ((#Mx_ET20 OR #Mx_ET21 OR #Mx_ET22 OR (((#Mx_ET02 AND NOT #PosTR_E1) OR #Mx_ET60 OR #Mx_ET61) AND ((#ConfigFB.Final_E2E4 AND #Selec_M4_Salida) OR (#ConfigFB.Inicio_E2E4 AND #Selec_M3_Salida))) OR (#Mx_ET02 AND #BloqueoActivo_OK AND NOT #PTF_MSal AND NOT #PosTR_E1) OR #Mx_ET180 OR #Mx_ET181 OR (#Mx_ET02 AND NOT #PosTR_E2 AND NOT #PosTR_E1) OR (NOT #PosTR_E1 AND (#CNTSeg_pHsMx_E1E3.CVU > 0) AND NOT #Selec_M2_Entrada AND NOT #Selec_M4_Entrada AND NOT #Selec_M2_Salida AND NOT #Selec_M4_Salida AND NOT #Mx_ET01) OR ((#Mx_ET90 OR #Mx_ET91) AND "ON") OR ((#Mx_ET40 OR #Mx_ET41 OR #Mx_ET43) AND "ON")) AND NOT "DB1_SalidasExterioresDeMesa".Mesa[#Mesa].Avanzar_E2E4 AND NOT "DB1_SalidasExterioresDeMesa".Mesa[#Mesa].Retroceder_E2E4) OR NOT #EstadoZona.Marcha_CBx OR #EstadoVI.Error_Mx OR #Error_Tx;
END_REGION

REGION Network 132: SALIDAS - Valor Frecuencia Lenta E2E4
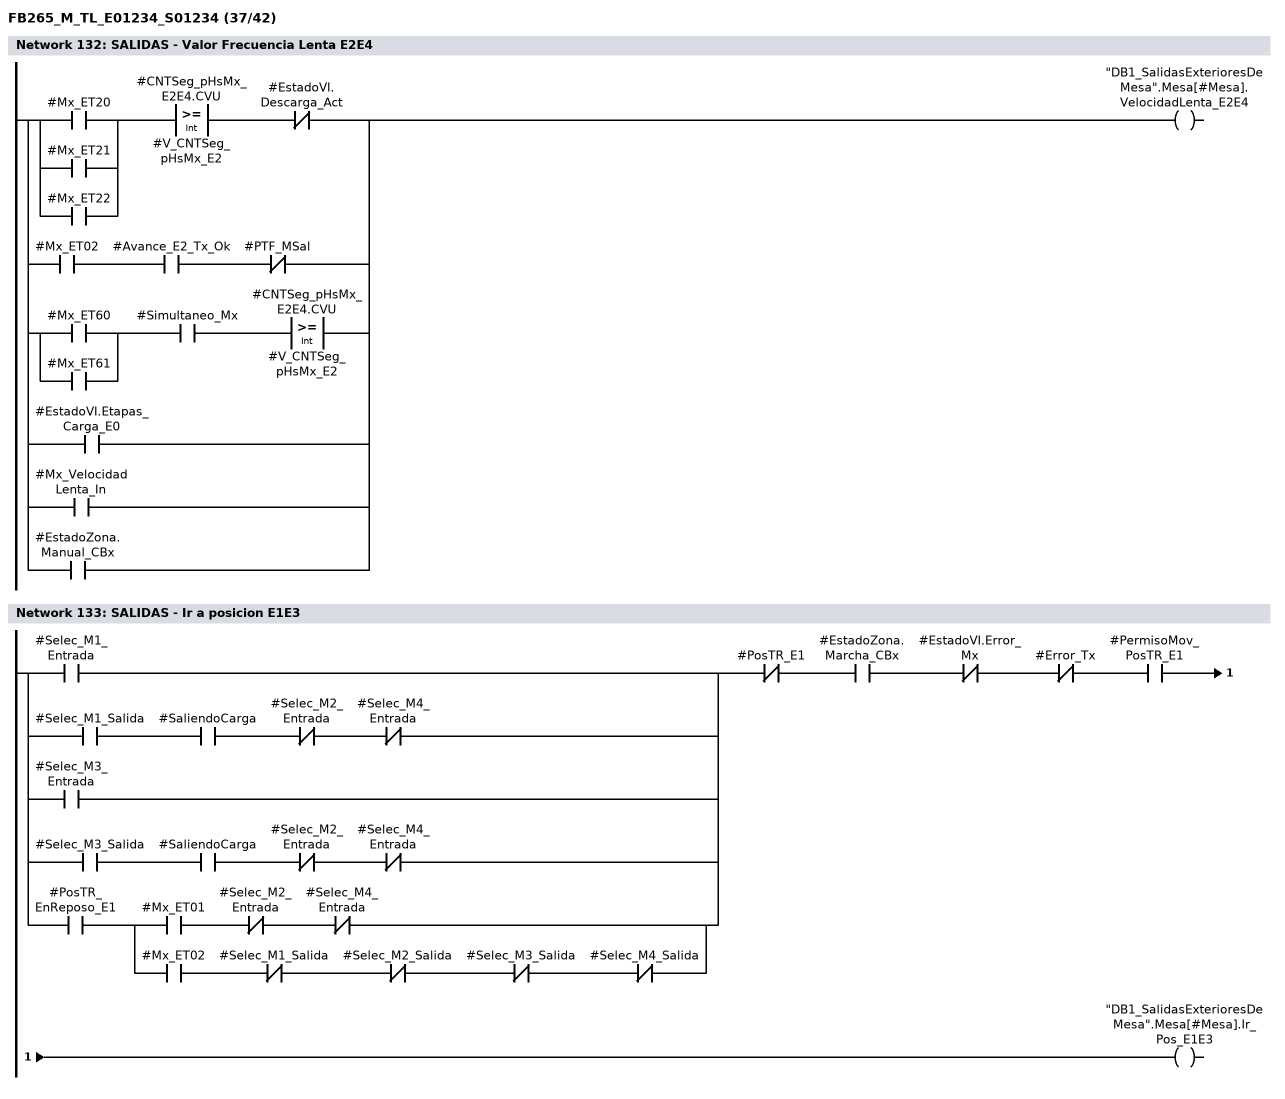
   RUNG wire#powerrail
      Contact( #Mx_ET20 )
      wire#w1
      { S7_Templates := "SrcType := Int" } GE_Contact(in1 := #CNTSeg_pHsMx_E2E4.CVU, in2 := #V_CNTSeg_pHsMx_E2)
      I_Contact( #EstadoVI.Descarga_Act )
      wire#w2
      Coil( "DB1_SalidasExterioresDeMesa".Mesa[#Mesa].VelocidadLenta_E2E4 )
   END_RUNG
   RUNG wire#powerrail
      Contact( #Mx_ET21 )
   END_RUNG wire#w1
   RUNG wire#powerrail
      Contact( #Mx_ET22 )
   END_RUNG wire#w1
   RUNG wire#powerrail
      Contact( #Mx_ET02 )
      Contact( #Avance_E2_Tx_Ok )
      I_Contact( #PTF_MSal )
   END_RUNG wire#w2
   RUNG wire#powerrail
      Contact( #Mx_ET60 )
      wire#w3
      Contact( #Simultaneo_Mx )
      { S7_Templates := "SrcType := Int" } GE_Contact(in1 := #CNTSeg_pHsMx_E2E4.CVU, in2 := #V_CNTSeg_pHsMx_E2)
   END_RUNG wire#w2
   RUNG wire#powerrail
      Contact( #Mx_ET61 )
   END_RUNG wire#w3
   RUNG wire#powerrail
      Contact( #EstadoVI.Etapas_Carga_E0 )
   END_RUNG wire#w2
   RUNG wire#powerrail
      Contact( #Mx_VelocidadLenta_In )
   END_RUNG wire#w2
   RUNG wire#powerrail
      Contact( #EstadoZona.Manual_CBx )
   END_RUNG wire#w2
   // the same network as SCL:
   "DB1_SalidasExterioresDeMesa".Mesa[#Mesa].VelocidadLenta_E2E4 := ((#Mx_ET20 OR #Mx_ET21 OR #Mx_ET22) AND (#CNTSeg_pHsMx_E2E4.CVU >= #V_CNTSeg_pHsMx_E2) AND NOT #EstadoVI.Descarga_Act) OR (#Mx_ET02 AND #Avance_E2_Tx_Ok AND NOT #PTF_MSal) OR ((#Mx_ET60 OR #Mx_ET61) AND #Simultaneo_Mx AND (#CNTSeg_pHsMx_E2E4.CVU >= #V_CNTSeg_pHsMx_E2)) OR #EstadoVI.Etapas_Carga_E0 OR #Mx_VelocidadLenta_In OR #EstadoZona.Manual_CBx;
END_REGION

REGION Network 133: SALIDAS - Ir a posicion E1E3
   RUNG wire#powerrail
      Contact( #Selec_M1_Entrada )
      wire#w1
      I_Contact( #PosTR_E1 )
      Contact( #EstadoZona.Marcha_CBx )
      I_Contact( #EstadoVI.Error_Mx )
      I_Contact( #Error_Tx )
      Contact( #PermisoMov_PosTR_E1 )
      Coil( "DB1_SalidasExterioresDeMesa".Mesa[#Mesa].Ir_Pos_E1E3 )
   END_RUNG
   RUNG wire#powerrail
      Contact( #Selec_M1_Salida )
      Contact( #SaliendoCarga )
      I_Contact( #Selec_M2_Entrada )
      I_Contact( #Selec_M4_Entrada )
   END_RUNG wire#w1
   RUNG wire#powerrail
      Contact( #Selec_M3_Entrada )
   END_RUNG wire#w1
   RUNG wire#powerrail
      Contact( #Selec_M3_Salida )
      Contact( #SaliendoCarga )
      I_Contact( #Selec_M2_Entrada )
      I_Contact( #Selec_M4_Entrada )
   END_RUNG wire#w1
   RUNG wire#powerrail
      Contact( #PosTR_EnReposo_E1 )
      wire#w2
      Contact( #Mx_ET01 )
      I_Contact( #Selec_M2_Entrada )
      I_Contact( #Selec_M4_Entrada )
   END_RUNG wire#w1
   RUNG wire#w2
      Contact( #Mx_ET02 )
      I_Contact( #Selec_M1_Salida )
      I_Contact( #Selec_M2_Salida )
      I_Contact( #Selec_M3_Salida )
      I_Contact( #Selec_M4_Salida )
   END_RUNG wire#w1
   // the same network as SCL:
   "DB1_SalidasExterioresDeMesa".Mesa[#Mesa].Ir_Pos_E1E3 := (#Selec_M1_Entrada OR (#Selec_M1_Salida AND #SaliendoCarga AND NOT #Selec_M2_Entrada AND NOT #Selec_M4_Entrada) OR #Selec_M3_Entrada OR (#Selec_M3_Salida AND #SaliendoCarga AND NOT #Selec_M2_Entrada AND NOT #Selec_M4_Entrada) OR (#PosTR_EnReposo_E1 AND ((#Mx_ET01 AND NOT #Selec_M2_Entrada AND NOT #Selec_M4_Entrada) OR (#Mx_ET02 AND NOT #Selec_M1_Salida AND NOT #Selec_M2_Salida AND NOT #Selec_M3_Salida AND NOT #Selec_M4_Salida)))) AND NOT #PosTR_E1 AND #EstadoZona.Marcha_CBx AND NOT #EstadoVI.Error_Mx AND NOT #Error_Tx AND #PermisoMov_PosTR_E1;
END_REGION

REGION Network 134: SALIDAS - Ir a posicion E2E4
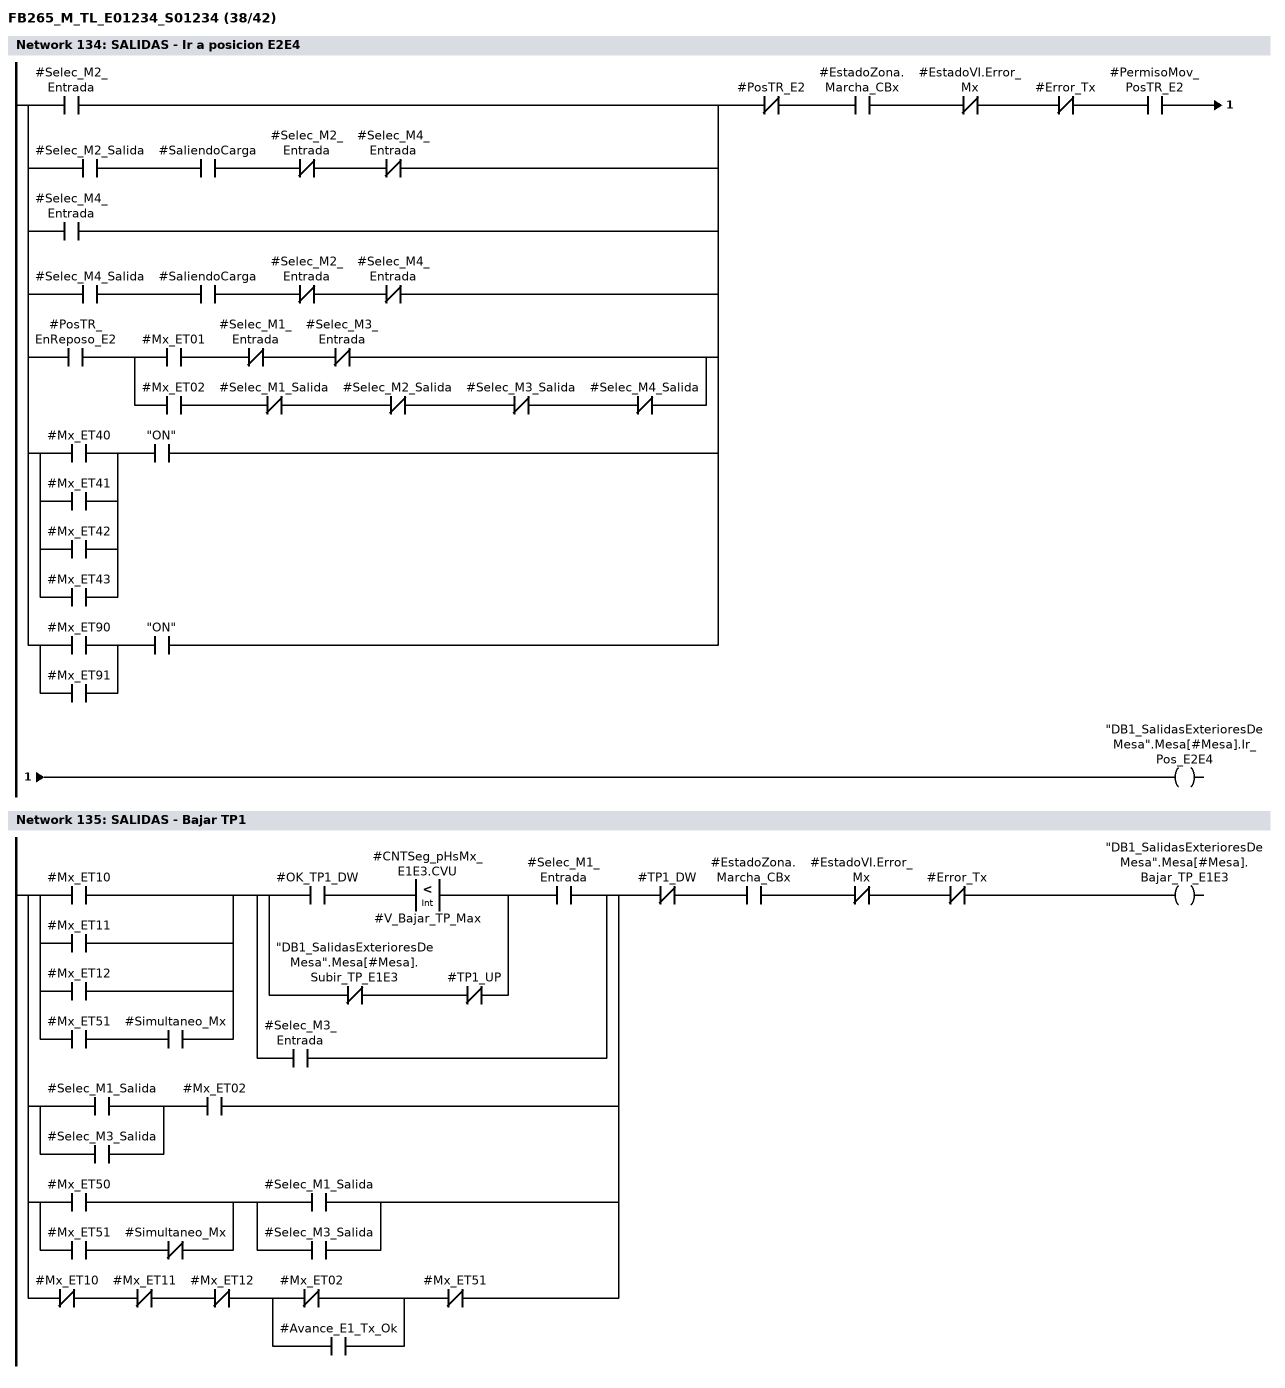
   RUNG wire#powerrail
      Contact( #Selec_M2_Entrada )
      wire#w1
      I_Contact( #PosTR_E2 )
      Contact( #EstadoZona.Marcha_CBx )
      I_Contact( #EstadoVI.Error_Mx )
      I_Contact( #Error_Tx )
      Contact( #PermisoMov_PosTR_E2 )
      Coil( "DB1_SalidasExterioresDeMesa".Mesa[#Mesa].Ir_Pos_E2E4 )
   END_RUNG
   RUNG wire#powerrail
      Contact( #Selec_M2_Salida )
      Contact( #SaliendoCarga )
      I_Contact( #Selec_M2_Entrada )
      I_Contact( #Selec_M4_Entrada )
   END_RUNG wire#w1
   RUNG wire#powerrail
      Contact( #Selec_M4_Entrada )
   END_RUNG wire#w1
   RUNG wire#powerrail
      Contact( #Selec_M4_Salida )
      Contact( #SaliendoCarga )
      I_Contact( #Selec_M2_Entrada )
      I_Contact( #Selec_M4_Entrada )
   END_RUNG wire#w1
   RUNG wire#powerrail
      Contact( #PosTR_EnReposo_E2 )
      wire#w2
      Contact( #Mx_ET01 )
      I_Contact( #Selec_M1_Entrada )
      I_Contact( #Selec_M3_Entrada )
   END_RUNG wire#w1
   RUNG wire#w2
      Contact( #Mx_ET02 )
      I_Contact( #Selec_M1_Salida )
      I_Contact( #Selec_M2_Salida )
      I_Contact( #Selec_M3_Salida )
      I_Contact( #Selec_M4_Salida )
   END_RUNG wire#w1
   RUNG wire#powerrail
      Contact( #Mx_ET40 )
      wire#w3
      Contact( "ON" )
   END_RUNG wire#w1
   RUNG wire#powerrail
      Contact( #Mx_ET41 )
   END_RUNG wire#w3
   RUNG wire#powerrail
      Contact( #Mx_ET42 )
   END_RUNG wire#w3
   RUNG wire#powerrail
      Contact( #Mx_ET43 )
   END_RUNG wire#w3
   RUNG wire#powerrail
      Contact( #Mx_ET90 )
      wire#w4
      Contact( "ON" )
   END_RUNG wire#w1
   RUNG wire#powerrail
      Contact( #Mx_ET91 )
   END_RUNG wire#w4
   // the same network as SCL:
   "DB1_SalidasExterioresDeMesa".Mesa[#Mesa].Ir_Pos_E2E4 := (#Selec_M2_Entrada OR (#Selec_M2_Salida AND #SaliendoCarga AND NOT #Selec_M2_Entrada AND NOT #Selec_M4_Entrada) OR #Selec_M4_Entrada OR (#Selec_M4_Salida AND #SaliendoCarga AND NOT #Selec_M2_Entrada AND NOT #Selec_M4_Entrada) OR (#PosTR_EnReposo_E2 AND ((#Mx_ET01 AND NOT #Selec_M1_Entrada AND NOT #Selec_M3_Entrada) OR (#Mx_ET02 AND NOT #Selec_M1_Salida AND NOT #Selec_M2_Salida AND NOT #Selec_M3_Salida AND NOT #Selec_M4_Salida))) OR ((#Mx_ET40 OR #Mx_ET41 OR #Mx_ET42 OR #Mx_ET43) AND "ON") OR ((#Mx_ET90 OR #Mx_ET91) AND "ON")) AND NOT #PosTR_E2 AND #EstadoZona.Marcha_CBx AND NOT #EstadoVI.Error_Mx AND NOT #Error_Tx AND #PermisoMov_PosTR_E2;
END_REGION

REGION Network 135: SALIDAS - Bajar TP1
   RUNG wire#powerrail
      Contact( #Mx_ET10 )
      wire#w1
      Contact( #OK_TP1_DW )
      { S7_Templates := "SrcType := Int" } LT_Contact(in1 := #CNTSeg_pHsMx_E1E3.CVU, in2 := #V_Bajar_TP_Max)
      wire#w2
      Contact( #Selec_M1_Entrada )
      wire#w3
      I_Contact( #TP1_DW )
      Contact( #EstadoZona.Marcha_CBx )
      I_Contact( #EstadoVI.Error_Mx )
      I_Contact( #Error_Tx )
      Coil( "DB1_SalidasExterioresDeMesa".Mesa[#Mesa].Bajar_TP_E1E3 )
   END_RUNG
   RUNG wire#powerrail
      Contact( #Mx_ET11 )
   END_RUNG wire#w1
   RUNG wire#powerrail
      Contact( #Mx_ET12 )
   END_RUNG wire#w1
   RUNG wire#powerrail
      Contact( #Mx_ET51 )
      Contact( #Simultaneo_Mx )
   END_RUNG wire#w1
   RUNG wire#w1
      I_Contact( "DB1_SalidasExterioresDeMesa".Mesa[#Mesa].Subir_TP_E1E3 )
      I_Contact( #TP1_UP )
   END_RUNG wire#w2
   RUNG wire#w1
      Contact( #Selec_M3_Entrada )
   END_RUNG wire#w3
   RUNG wire#powerrail
      Contact( #Selec_M1_Salida )
      wire#w4
      Contact( #Mx_ET02 )
   END_RUNG wire#w3
   RUNG wire#powerrail
      Contact( #Selec_M3_Salida )
   END_RUNG wire#w4
   RUNG wire#powerrail
      Contact( #Mx_ET50 )
      wire#w5
      Contact( #Selec_M1_Salida )
   END_RUNG wire#w3
   RUNG wire#powerrail
      Contact( #Mx_ET51 )
      I_Contact( #Simultaneo_Mx )
   END_RUNG wire#w5
   RUNG wire#w5
      Contact( #Selec_M3_Salida )
   END_RUNG wire#w3
   RUNG wire#powerrail
      I_Contact( #Mx_ET10 )
      I_Contact( #Mx_ET11 )
      I_Contact( #Mx_ET12 )
      wire#w6
      I_Contact( #Mx_ET02 )
      wire#w7
      I_Contact( #Mx_ET51 )
   END_RUNG wire#w3
   RUNG wire#w6
      Contact( #Avance_E1_Tx_Ok )
   END_RUNG wire#w7
   // the same network as SCL:
   "DB1_SalidasExterioresDeMesa".Mesa[#Mesa].Bajar_TP_E1E3 := (((#Mx_ET10 OR #Mx_ET11 OR #Mx_ET12 OR (#Mx_ET51 AND #Simultaneo_Mx)) AND ((((#OK_TP1_DW AND (#CNTSeg_pHsMx_E1E3.CVU < #V_Bajar_TP_Max)) OR (NOT "DB1_SalidasExterioresDeMesa".Mesa[#Mesa].Subir_TP_E1E3 AND NOT #TP1_UP)) AND #Selec_M1_Entrada) OR #Selec_M3_Entrada)) OR ((#Selec_M1_Salida OR #Selec_M3_Salida) AND #Mx_ET02) OR ((#Mx_ET50 OR (#Mx_ET51 AND NOT #Simultaneo_Mx)) AND (#Selec_M1_Salida OR #Selec_M3_Salida)) OR (NOT #Mx_ET10 AND NOT #Mx_ET11 AND NOT #Mx_ET12 AND (NOT #Mx_ET02 OR #Avance_E1_Tx_Ok) AND NOT #Mx_ET51)) AND NOT #TP1_DW AND #EstadoZona.Marcha_CBx AND NOT #EstadoVI.Error_Mx AND NOT #Error_Tx;
END_REGION

REGION Network 136: SALIDAS - Subir TP1
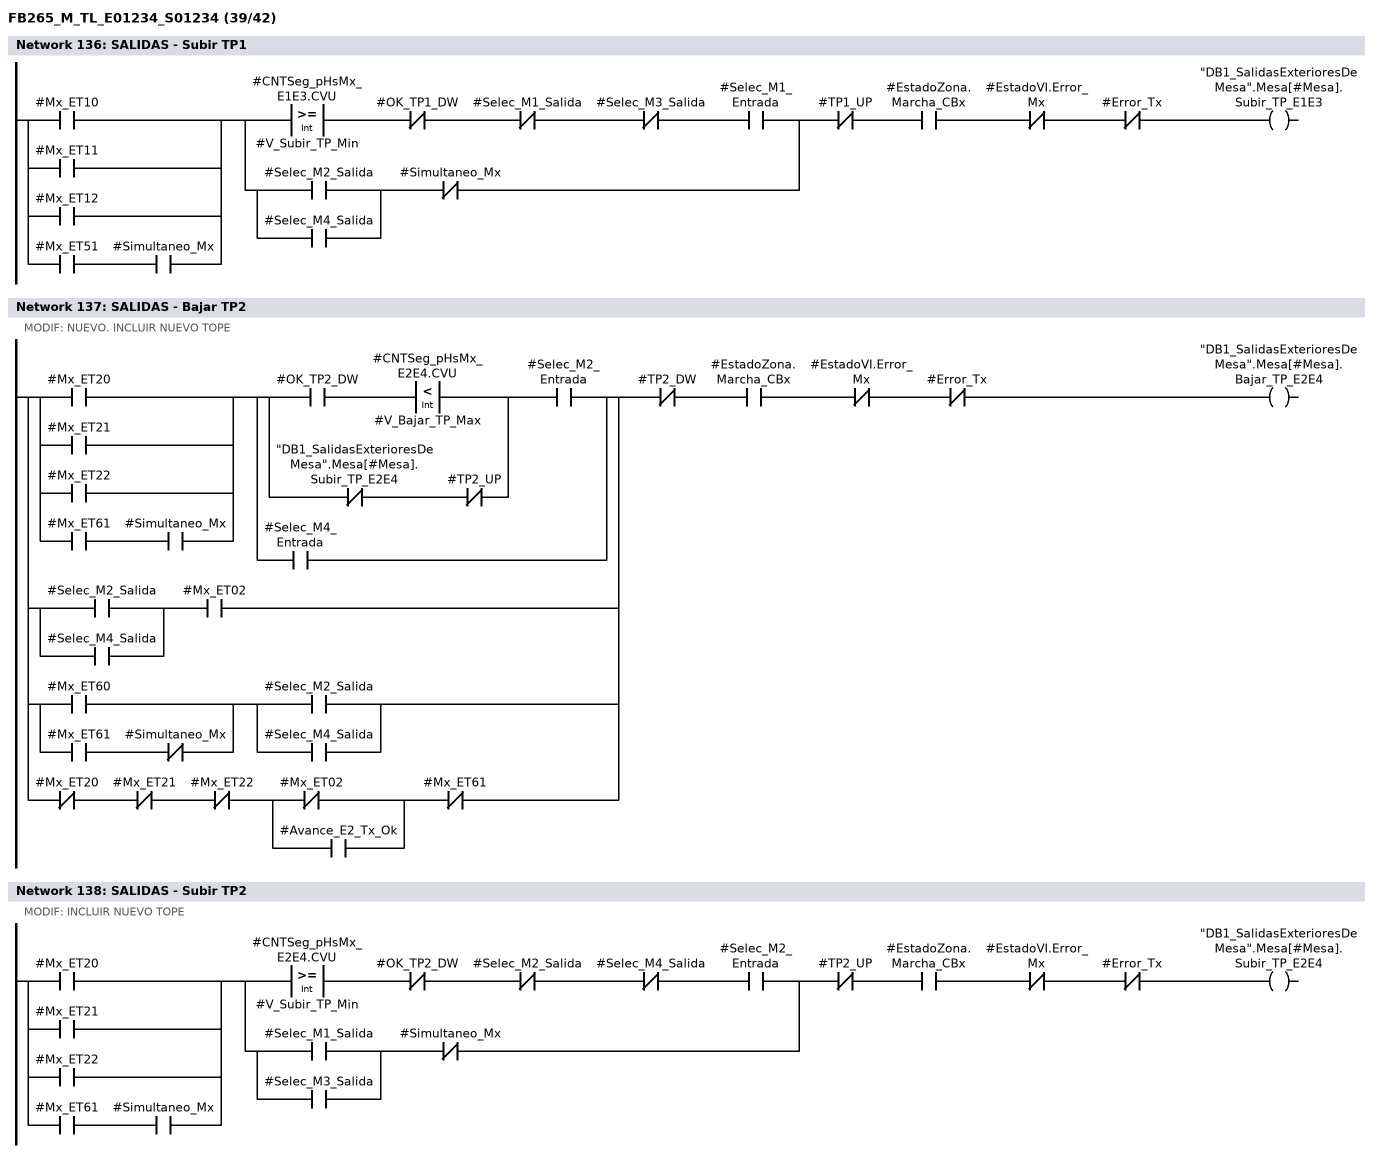
   RUNG wire#powerrail
      Contact( #Mx_ET10 )
      wire#w1
      { S7_Templates := "SrcType := Int" } GE_Contact(in1 := #CNTSeg_pHsMx_E1E3.CVU, in2 := #V_Subir_TP_Min)
      I_Contact( #OK_TP1_DW )
      I_Contact( #Selec_M1_Salida )
      I_Contact( #Selec_M3_Salida )
      Contact( #Selec_M1_Entrada )
      wire#w2
      I_Contact( #TP1_UP )
      Contact( #EstadoZona.Marcha_CBx )
      I_Contact( #EstadoVI.Error_Mx )
      I_Contact( #Error_Tx )
      Coil( "DB1_SalidasExterioresDeMesa".Mesa[#Mesa].Subir_TP_E1E3 )
   END_RUNG
   RUNG wire#powerrail
      Contact( #Mx_ET11 )
   END_RUNG wire#w1
   RUNG wire#powerrail
      Contact( #Mx_ET12 )
   END_RUNG wire#w1
   RUNG wire#powerrail
      Contact( #Mx_ET51 )
      Contact( #Simultaneo_Mx )
   END_RUNG wire#w1
   RUNG wire#w1
      Contact( #Selec_M2_Salida )
      wire#w3
      I_Contact( #Simultaneo_Mx )
   END_RUNG wire#w2
   RUNG wire#w1
      Contact( #Selec_M4_Salida )
   END_RUNG wire#w3
   // the same network as SCL:
   "DB1_SalidasExterioresDeMesa".Mesa[#Mesa].Subir_TP_E1E3 := (#Mx_ET10 OR #Mx_ET11 OR #Mx_ET12 OR (#Mx_ET51 AND #Simultaneo_Mx)) AND (((#CNTSeg_pHsMx_E1E3.CVU >= #V_Subir_TP_Min) AND NOT #OK_TP1_DW AND NOT #Selec_M1_Salida AND NOT #Selec_M3_Salida AND #Selec_M1_Entrada) OR ((#Selec_M2_Salida OR #Selec_M4_Salida) AND NOT #Simultaneo_Mx)) AND NOT #TP1_UP AND #EstadoZona.Marcha_CBx AND NOT #EstadoVI.Error_Mx AND NOT #Error_Tx;
END_REGION

REGION Network 137: SALIDAS - Bajar TP2
   // MODIF: NUEVO. INCLUIR NUEVO TOPE
   RUNG wire#powerrail
      Contact( #Mx_ET20 )
      wire#w1
      Contact( #OK_TP2_DW )
      { S7_Templates := "SrcType := Int" } LT_Contact(in1 := #CNTSeg_pHsMx_E2E4.CVU, in2 := #V_Bajar_TP_Max)
      wire#w2
      Contact( #Selec_M2_Entrada )
      wire#w3
      I_Contact( #TP2_DW )
      Contact( #EstadoZona.Marcha_CBx )
      I_Contact( #EstadoVI.Error_Mx )
      I_Contact( #Error_Tx )
      Coil( "DB1_SalidasExterioresDeMesa".Mesa[#Mesa].Bajar_TP_E2E4 )
   END_RUNG
   RUNG wire#powerrail
      Contact( #Mx_ET21 )
   END_RUNG wire#w1
   RUNG wire#powerrail
      Contact( #Mx_ET22 )
   END_RUNG wire#w1
   RUNG wire#powerrail
      Contact( #Mx_ET61 )
      Contact( #Simultaneo_Mx )
   END_RUNG wire#w1
   RUNG wire#w1
      I_Contact( "DB1_SalidasExterioresDeMesa".Mesa[#Mesa].Subir_TP_E2E4 )
      I_Contact( #TP2_UP )
   END_RUNG wire#w2
   RUNG wire#w1
      Contact( #Selec_M4_Entrada )
   END_RUNG wire#w3
   RUNG wire#powerrail
      Contact( #Selec_M2_Salida )
      wire#w4
      Contact( #Mx_ET02 )
   END_RUNG wire#w3
   RUNG wire#powerrail
      Contact( #Selec_M4_Salida )
   END_RUNG wire#w4
   RUNG wire#powerrail
      Contact( #Mx_ET60 )
      wire#w5
      Contact( #Selec_M2_Salida )
   END_RUNG wire#w3
   RUNG wire#powerrail
      Contact( #Mx_ET61 )
      I_Contact( #Simultaneo_Mx )
   END_RUNG wire#w5
   RUNG wire#w5
      Contact( #Selec_M4_Salida )
   END_RUNG wire#w3
   RUNG wire#powerrail
      I_Contact( #Mx_ET20 )
      I_Contact( #Mx_ET21 )
      I_Contact( #Mx_ET22 )
      wire#w6
      I_Contact( #Mx_ET02 )
      wire#w7
      I_Contact( #Mx_ET61 )
   END_RUNG wire#w3
   RUNG wire#w6
      Contact( #Avance_E2_Tx_Ok )
   END_RUNG wire#w7
   // the same network as SCL:
   "DB1_SalidasExterioresDeMesa".Mesa[#Mesa].Bajar_TP_E2E4 := (((#Mx_ET20 OR #Mx_ET21 OR #Mx_ET22 OR (#Mx_ET61 AND #Simultaneo_Mx)) AND ((((#OK_TP2_DW AND (#CNTSeg_pHsMx_E2E4.CVU < #V_Bajar_TP_Max)) OR (NOT "DB1_SalidasExterioresDeMesa".Mesa[#Mesa].Subir_TP_E2E4 AND NOT #TP2_UP)) AND #Selec_M2_Entrada) OR #Selec_M4_Entrada)) OR ((#Selec_M2_Salida OR #Selec_M4_Salida) AND #Mx_ET02) OR ((#Mx_ET60 OR (#Mx_ET61 AND NOT #Simultaneo_Mx)) AND (#Selec_M2_Salida OR #Selec_M4_Salida)) OR (NOT #Mx_ET20 AND NOT #Mx_ET21 AND NOT #Mx_ET22 AND (NOT #Mx_ET02 OR #Avance_E2_Tx_Ok) AND NOT #Mx_ET61)) AND NOT #TP2_DW AND #EstadoZona.Marcha_CBx AND NOT #EstadoVI.Error_Mx AND NOT #Error_Tx;
END_REGION

REGION Network 138: SALIDAS - Subir TP2
   // MODIF: INCLUIR NUEVO TOPE
   RUNG wire#powerrail
      Contact( #Mx_ET20 )
      wire#w1
      { S7_Templates := "SrcType := Int" } GE_Contact(in1 := #CNTSeg_pHsMx_E2E4.CVU, in2 := #V_Subir_TP_Min)
      I_Contact( #OK_TP2_DW )
      I_Contact( #Selec_M2_Salida )
      I_Contact( #Selec_M4_Salida )
      Contact( #Selec_M2_Entrada )
      wire#w2
      I_Contact( #TP2_UP )
      Contact( #EstadoZona.Marcha_CBx )
      I_Contact( #EstadoVI.Error_Mx )
      I_Contact( #Error_Tx )
      Coil( "DB1_SalidasExterioresDeMesa".Mesa[#Mesa].Subir_TP_E2E4 )
   END_RUNG
   RUNG wire#powerrail
      Contact( #Mx_ET21 )
   END_RUNG wire#w1
   RUNG wire#powerrail
      Contact( #Mx_ET22 )
   END_RUNG wire#w1
   RUNG wire#powerrail
      Contact( #Mx_ET61 )
      Contact( #Simultaneo_Mx )
   END_RUNG wire#w1
   RUNG wire#w1
      Contact( #Selec_M1_Salida )
      wire#w3
      I_Contact( #Simultaneo_Mx )
   END_RUNG wire#w2
   RUNG wire#w1
      Contact( #Selec_M3_Salida )
   END_RUNG wire#w3
   // the same network as SCL:
   "DB1_SalidasExterioresDeMesa".Mesa[#Mesa].Subir_TP_E2E4 := (#Mx_ET20 OR #Mx_ET21 OR #Mx_ET22 OR (#Mx_ET61 AND #Simultaneo_Mx)) AND (((#CNTSeg_pHsMx_E2E4.CVU >= #V_Subir_TP_Min) AND NOT #OK_TP2_DW AND NOT #Selec_M2_Salida AND NOT #Selec_M4_Salida AND #Selec_M2_Entrada) OR ((#Selec_M1_Salida OR #Selec_M3_Salida) AND NOT #Simultaneo_Mx)) AND NOT #TP2_UP AND #EstadoZona.Marcha_CBx AND NOT #EstadoVI.Error_Mx AND NOT #Error_Tx;
END_REGION

REGION Network 139: ESTADOS DE LA MESA
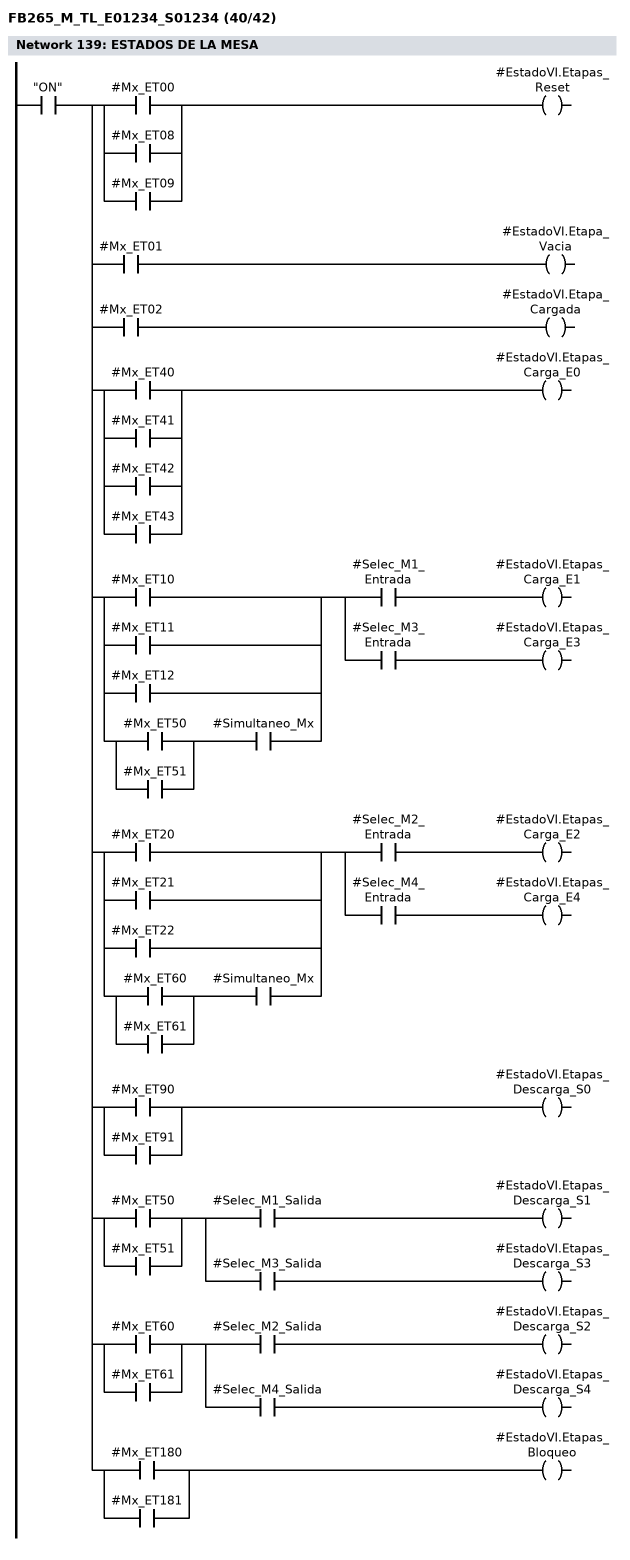
   RUNG wire#powerrail
      Contact( "ON" )
      wire#w1
      Contact( #Mx_ET00 )
      wire#w2
      Coil( #EstadoVI.Etapas_Reset )
   END_RUNG
   RUNG wire#w1
      Contact( #Mx_ET08 )
   END_RUNG wire#w2
   RUNG wire#w1
      Contact( #Mx_ET09 )
   END_RUNG wire#w2
   RUNG wire#w1
      Contact( #Mx_ET01 )
      Coil( #EstadoVI.Etapa_Vacia )
   END_RUNG
   RUNG wire#w1
      Contact( #Mx_ET02 )
      Coil( #EstadoVI.Etapa_Cargada )
   END_RUNG
   RUNG wire#w1
      Contact( #Mx_ET40 )
      wire#w3
      Coil( #EstadoVI.Etapas_Carga_E0 )
   END_RUNG
   RUNG wire#w1
      Contact( #Mx_ET41 )
   END_RUNG wire#w3
   RUNG wire#w1
      Contact( #Mx_ET42 )
   END_RUNG wire#w3
   RUNG wire#w1
      Contact( #Mx_ET43 )
   END_RUNG wire#w3
   RUNG wire#w1
      Contact( #Mx_ET10 )
      wire#w4
      Contact( #Selec_M1_Entrada )
      Coil( #EstadoVI.Etapas_Carga_E1 )
   END_RUNG
   RUNG wire#w1
      Contact( #Mx_ET11 )
   END_RUNG wire#w4
   RUNG wire#w1
      Contact( #Mx_ET12 )
   END_RUNG wire#w4
   RUNG wire#w1
      Contact( #Mx_ET50 )
      wire#w5
      Contact( #Simultaneo_Mx )
   END_RUNG wire#w4
   RUNG wire#w1
      Contact( #Mx_ET51 )
   END_RUNG wire#w5
   RUNG wire#w4
      Contact( #Selec_M3_Entrada )
      Coil( #EstadoVI.Etapas_Carga_E3 )
   END_RUNG
   RUNG wire#w1
      Contact( #Mx_ET20 )
      wire#w6
      Contact( #Selec_M2_Entrada )
      Coil( #EstadoVI.Etapas_Carga_E2 )
   END_RUNG
   RUNG wire#w1
      Contact( #Mx_ET21 )
   END_RUNG wire#w6
   RUNG wire#w1
      Contact( #Mx_ET22 )
   END_RUNG wire#w6
   RUNG wire#w1
      Contact( #Mx_ET60 )
      wire#w7
      Contact( #Simultaneo_Mx )
   END_RUNG wire#w6
   RUNG wire#w1
      Contact( #Mx_ET61 )
   END_RUNG wire#w7
   RUNG wire#w6
      Contact( #Selec_M4_Entrada )
      Coil( #EstadoVI.Etapas_Carga_E4 )
   END_RUNG
   RUNG wire#w1
      Contact( #Mx_ET90 )
      wire#w8
      Coil( #EstadoVI.Etapas_Descarga_S0 )
   END_RUNG
   RUNG wire#w1
      Contact( #Mx_ET91 )
   END_RUNG wire#w8
   RUNG wire#w1
      Contact( #Mx_ET50 )
      wire#w9
      Contact( #Selec_M1_Salida )
      Coil( #EstadoVI.Etapas_Descarga_S1 )
   END_RUNG
   RUNG wire#w1
      Contact( #Mx_ET51 )
   END_RUNG wire#w9
   RUNG wire#w9
      Contact( #Selec_M3_Salida )
      Coil( #EstadoVI.Etapas_Descarga_S3 )
   END_RUNG
   RUNG wire#w1
      Contact( #Mx_ET60 )
      wire#w10
      Contact( #Selec_M2_Salida )
      Coil( #EstadoVI.Etapas_Descarga_S2 )
   END_RUNG
   RUNG wire#w1
      Contact( #Mx_ET61 )
   END_RUNG wire#w10
   RUNG wire#w10
      Contact( #Selec_M4_Salida )
      Coil( #EstadoVI.Etapas_Descarga_S4 )
   END_RUNG
   RUNG wire#w1
      Contact( #Mx_ET180 )
      wire#w11
      Coil( #EstadoVI.Etapas_Bloqueo )
   END_RUNG
   RUNG wire#w1
      Contact( #Mx_ET181 )
   END_RUNG wire#w11
   // the same network as SCL:
   #EstadoVI.Etapas_Reset := "ON" AND (#Mx_ET00 OR #Mx_ET08 OR #Mx_ET09);
   #EstadoVI.Etapa_Vacia := "ON" AND #Mx_ET01;
   #EstadoVI.Etapa_Cargada := "ON" AND #Mx_ET02;
   #EstadoVI.Etapas_Carga_E0 := "ON" AND (#Mx_ET40 OR #Mx_ET41 OR #Mx_ET42 OR #Mx_ET43);
   #_w1 := "ON" AND (#Mx_ET10 OR #Mx_ET11 OR #Mx_ET12 OR ((#Mx_ET50 OR #Mx_ET51) AND #Simultaneo_Mx));
   #EstadoVI.Etapas_Carga_E1 := #_w1 AND #Selec_M1_Entrada;
   #EstadoVI.Etapas_Carga_E3 := #_w1 AND #Selec_M3_Entrada;
   #_w2 := "ON" AND (#Mx_ET20 OR #Mx_ET21 OR #Mx_ET22 OR ((#Mx_ET60 OR #Mx_ET61) AND #Simultaneo_Mx));
   #EstadoVI.Etapas_Carga_E2 := #_w2 AND #Selec_M2_Entrada;
   #EstadoVI.Etapas_Carga_E4 := #_w2 AND #Selec_M4_Entrada;
   #EstadoVI.Etapas_Descarga_S0 := "ON" AND (#Mx_ET90 OR #Mx_ET91);
   #_w3 := "ON" AND (#Mx_ET50 OR #Mx_ET51);
   #EstadoVI.Etapas_Descarga_S1 := #_w3 AND #Selec_M1_Salida;
   #EstadoVI.Etapas_Descarga_S3 := #_w3 AND #Selec_M3_Salida;
   #_w4 := "ON" AND (#Mx_ET60 OR #Mx_ET61);
   #EstadoVI.Etapas_Descarga_S2 := #_w4 AND #Selec_M2_Salida;
   #EstadoVI.Etapas_Descarga_S4 := #_w4 AND #Selec_M4_Salida;
   #EstadoVI.Etapas_Bloqueo := "ON" AND (#Mx_ET180 OR #Mx_ET181);
END_REGION

REGION Network 140: ENTRADAS DE LA MESA
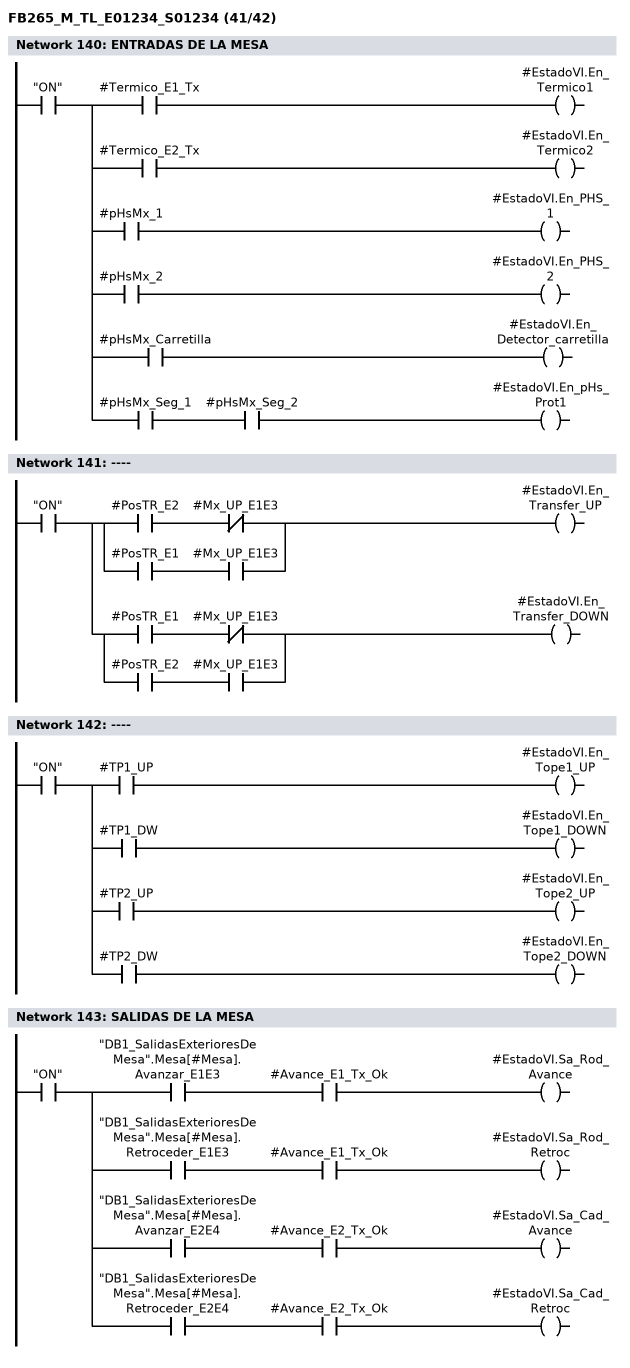
   RUNG wire#powerrail
      Contact( "ON" )
      wire#w1
      Contact( #Termico_E1_Tx )
      Coil( #EstadoVI.En_Termico1 )
   END_RUNG
   RUNG wire#w1
      Contact( #Termico_E2_Tx )
      Coil( #EstadoVI.En_Termico2 )
   END_RUNG
   RUNG wire#w1
      Contact( #pHsMx_1 )
      Coil( #EstadoVI.En_PHS_1 )
   END_RUNG
   RUNG wire#w1
      Contact( #pHsMx_2 )
      Coil( #EstadoVI.En_PHS_2 )
   END_RUNG
   RUNG wire#w1
      Contact( #pHsMx_Carretilla )
      Coil( #EstadoVI.En_Detector_carretilla )
   END_RUNG
   RUNG wire#w1
      Contact( #pHsMx_Seg_1 )
      Contact( #pHsMx_Seg_2 )
      Coil( #EstadoVI.En_pHs_Prot1 )
   END_RUNG
   // the same network as SCL:
   #EstadoVI.En_Termico1 := "ON" AND #Termico_E1_Tx;
   #EstadoVI.En_Termico2 := "ON" AND #Termico_E2_Tx;
   #EstadoVI.En_PHS_1 := "ON" AND #pHsMx_1;
   #EstadoVI.En_PHS_2 := "ON" AND #pHsMx_2;
   #EstadoVI.En_Detector_carretilla := "ON" AND #pHsMx_Carretilla;
   #EstadoVI.En_pHs_Prot1 := "ON" AND #pHsMx_Seg_1 AND #pHsMx_Seg_2;
END_REGION

REGION Network 141: ----
   RUNG wire#powerrail
      Contact( "ON" )
      wire#w1
      Contact( #PosTR_E2 )
      I_Contact( #Mx_UP_E1E3 )
      wire#w2
      Coil( #EstadoVI.En_Transfer_UP )
   END_RUNG
   RUNG wire#w1
      Contact( #PosTR_E1 )
      Contact( #Mx_UP_E1E3 )
   END_RUNG wire#w2
   RUNG wire#w1
      Contact( #PosTR_E1 )
      I_Contact( #Mx_UP_E1E3 )
      wire#w3
      Coil( #EstadoVI.En_Transfer_DOWN )
   END_RUNG
   RUNG wire#w1
      Contact( #PosTR_E2 )
      Contact( #Mx_UP_E1E3 )
   END_RUNG wire#w3
   // the same network as SCL:
   #EstadoVI.En_Transfer_UP := "ON" AND ((#PosTR_E2 AND NOT #Mx_UP_E1E3) OR (#PosTR_E1 AND #Mx_UP_E1E3));
   #EstadoVI.En_Transfer_DOWN := "ON" AND ((#PosTR_E1 AND NOT #Mx_UP_E1E3) OR (#PosTR_E2 AND #Mx_UP_E1E3));
END_REGION

REGION Network 142: ----
   RUNG wire#powerrail
      Contact( "ON" )
      wire#w1
      Contact( #TP1_UP )
      Coil( #EstadoVI.En_Tope1_UP )
   END_RUNG
   RUNG wire#w1
      Contact( #TP1_DW )
      Coil( #EstadoVI.En_Tope1_DOWN )
   END_RUNG
   RUNG wire#w1
      Contact( #TP2_UP )
      Coil( #EstadoVI.En_Tope2_UP )
   END_RUNG
   RUNG wire#w1
      Contact( #TP2_DW )
      Coil( #EstadoVI.En_Tope2_DOWN )
   END_RUNG
   // the same network as SCL:
   #EstadoVI.En_Tope1_UP := "ON" AND #TP1_UP;
   #EstadoVI.En_Tope1_DOWN := "ON" AND #TP1_DW;
   #EstadoVI.En_Tope2_UP := "ON" AND #TP2_UP;
   #EstadoVI.En_Tope2_DOWN := "ON" AND #TP2_DW;
END_REGION

REGION Network 143: SALIDAS DE LA MESA
   RUNG wire#powerrail
      Contact( "ON" )
      wire#w1
      Contact( "DB1_SalidasExterioresDeMesa".Mesa[#Mesa].Avanzar_E1E3 )
      Contact( #Avance_E1_Tx_Ok )
      Coil( #EstadoVI.Sa_Rod_Avance )
   END_RUNG
   RUNG wire#w1
      Contact( "DB1_SalidasExterioresDeMesa".Mesa[#Mesa].Retroceder_E1E3 )
      Contact( #Avance_E1_Tx_Ok )
      Coil( #EstadoVI.Sa_Rod_Retroc )
   END_RUNG
   RUNG wire#w1
      Contact( "DB1_SalidasExterioresDeMesa".Mesa[#Mesa].Avanzar_E2E4 )
      Contact( #Avance_E2_Tx_Ok )
      Coil( #EstadoVI.Sa_Cad_Avance )
   END_RUNG
   RUNG wire#w1
      Contact( "DB1_SalidasExterioresDeMesa".Mesa[#Mesa].Retroceder_E2E4 )
      Contact( #Avance_E2_Tx_Ok )
      Coil( #EstadoVI.Sa_Cad_Retroc )
   END_RUNG
   // the same network as SCL:
   #EstadoVI.Sa_Rod_Avance := "ON" AND "DB1_SalidasExterioresDeMesa".Mesa[#Mesa].Avanzar_E1E3 AND #Avance_E1_Tx_Ok;
   #EstadoVI.Sa_Rod_Retroc := "ON" AND "DB1_SalidasExterioresDeMesa".Mesa[#Mesa].Retroceder_E1E3 AND #Avance_E1_Tx_Ok;
   #EstadoVI.Sa_Cad_Avance := "ON" AND "DB1_SalidasExterioresDeMesa".Mesa[#Mesa].Avanzar_E2E4 AND #Avance_E2_Tx_Ok;
   #EstadoVI.Sa_Cad_Retroc := "ON" AND "DB1_SalidasExterioresDeMesa".Mesa[#Mesa].Retroceder_E2E4 AND #Avance_E2_Tx_Ok;
END_REGION

REGION Network 144: ----
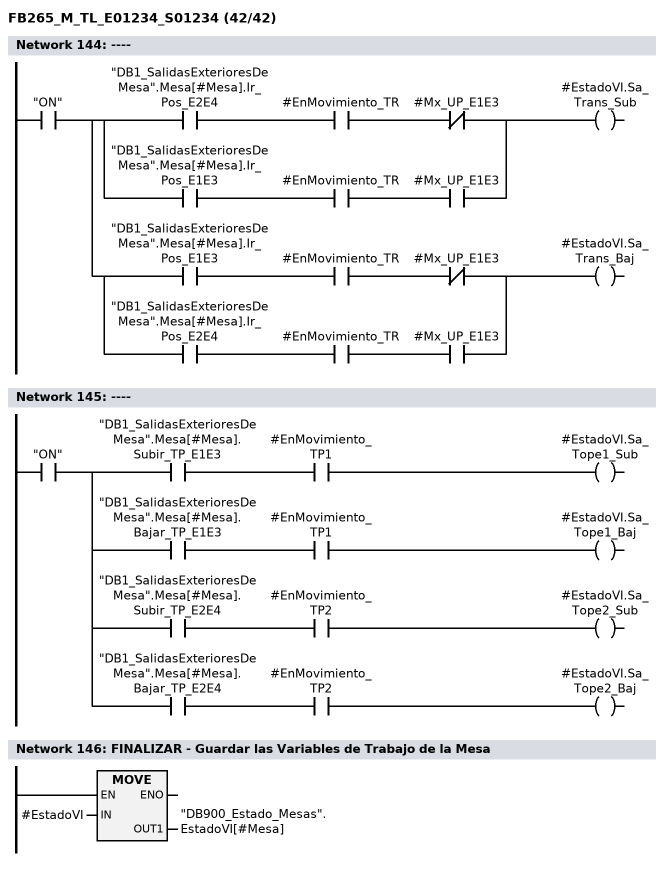
   RUNG wire#powerrail
      Contact( "ON" )
      wire#w1
      Contact( "DB1_SalidasExterioresDeMesa".Mesa[#Mesa].Ir_Pos_E2E4 )
      Contact( #EnMovimiento_TR )
      I_Contact( #Mx_UP_E1E3 )
      wire#w2
      Coil( #EstadoVI.Sa_Trans_Sub )
   END_RUNG
   RUNG wire#w1
      Contact( "DB1_SalidasExterioresDeMesa".Mesa[#Mesa].Ir_Pos_E1E3 )
      Contact( #EnMovimiento_TR )
      Contact( #Mx_UP_E1E3 )
   END_RUNG wire#w2
   RUNG wire#w1
      Contact( "DB1_SalidasExterioresDeMesa".Mesa[#Mesa].Ir_Pos_E1E3 )
      Contact( #EnMovimiento_TR )
      I_Contact( #Mx_UP_E1E3 )
      wire#w3
      Coil( #EstadoVI.Sa_Trans_Baj )
   END_RUNG
   RUNG wire#w1
      Contact( "DB1_SalidasExterioresDeMesa".Mesa[#Mesa].Ir_Pos_E2E4 )
      Contact( #EnMovimiento_TR )
      Contact( #Mx_UP_E1E3 )
   END_RUNG wire#w3
   // the same network as SCL:
   #EstadoVI.Sa_Trans_Sub := "ON" AND (("DB1_SalidasExterioresDeMesa".Mesa[#Mesa].Ir_Pos_E2E4 AND #EnMovimiento_TR AND NOT #Mx_UP_E1E3) OR ("DB1_SalidasExterioresDeMesa".Mesa[#Mesa].Ir_Pos_E1E3 AND #EnMovimiento_TR AND #Mx_UP_E1E3));
   #EstadoVI.Sa_Trans_Baj := "ON" AND (("DB1_SalidasExterioresDeMesa".Mesa[#Mesa].Ir_Pos_E1E3 AND #EnMovimiento_TR AND NOT #Mx_UP_E1E3) OR ("DB1_SalidasExterioresDeMesa".Mesa[#Mesa].Ir_Pos_E2E4 AND #EnMovimiento_TR AND #Mx_UP_E1E3));
END_REGION

REGION Network 145: ----
   RUNG wire#powerrail
      Contact( "ON" )
      wire#w1
      Contact( "DB1_SalidasExterioresDeMesa".Mesa[#Mesa].Subir_TP_E1E3 )
      Contact( #EnMovimiento_TP1 )
      Coil( #EstadoVI.Sa_Tope1_Sub )
   END_RUNG
   RUNG wire#w1
      Contact( "DB1_SalidasExterioresDeMesa".Mesa[#Mesa].Bajar_TP_E1E3 )
      Contact( #EnMovimiento_TP1 )
      Coil( #EstadoVI.Sa_Tope1_Baj )
   END_RUNG
   RUNG wire#w1
      Contact( "DB1_SalidasExterioresDeMesa".Mesa[#Mesa].Subir_TP_E2E4 )
      Contact( #EnMovimiento_TP2 )
      Coil( #EstadoVI.Sa_Tope2_Sub )
   END_RUNG
   RUNG wire#w1
      Contact( "DB1_SalidasExterioresDeMesa".Mesa[#Mesa].Bajar_TP_E2E4 )
      Contact( #EnMovimiento_TP2 )
      Coil( #EstadoVI.Sa_Tope2_Baj )
   END_RUNG
   // the same network as SCL:
   #EstadoVI.Sa_Tope1_Sub := "ON" AND "DB1_SalidasExterioresDeMesa".Mesa[#Mesa].Subir_TP_E1E3 AND #EnMovimiento_TP1;
   #EstadoVI.Sa_Tope1_Baj := "ON" AND "DB1_SalidasExterioresDeMesa".Mesa[#Mesa].Bajar_TP_E1E3 AND #EnMovimiento_TP1;
   #EstadoVI.Sa_Tope2_Sub := "ON" AND "DB1_SalidasExterioresDeMesa".Mesa[#Mesa].Subir_TP_E2E4 AND #EnMovimiento_TP2;
   #EstadoVI.Sa_Tope2_Baj := "ON" AND "DB1_SalidasExterioresDeMesa".Mesa[#Mesa].Bajar_TP_E2E4 AND #EnMovimiento_TP2;
END_REGION

REGION Network 146: FINALIZAR - Guardar las Variables de Trabajo de la Mesa
   RUNG wire#powerrail
      Move(in := #EstadoVI, out1 => "DB900_Estado_Mesas".EstadoVI[#Mesa])
   END_RUNG
   // the same network as SCL:
   "DB900_Estado_Mesas".EstadoVI[#Mesa] := #EstadoVI;
END_REGION
END_FUNCTION_BLOCK
